LIN {X 0,Y 158.907,Z 446.881,A -85,B 0,C 180,E1 -23891.248,E2 -23891.248} C_VEL
LIN {X 0,Y 155.468,Z 440.852,A -85,B 0,C 180,E1 -23892.757,E2 -23892.757} C_VEL
LIN {X 0,Y 153.776,Z 436.815,A -85,B 0,C 180,E1 -23893.575,E2 -23893.575} C_VEL
LIN {X 0,Y 152.527,Z 433.767,A -85,B 0,C 180,E1 -23894.17,E2 -23894.17} C_VEL
LIN {X 0,Y 152.355,Z 432.875,A -85,B 0,C 180,E1 -23894.389,E2 -23894.389} C_VEL
LIN {X 0,Y 151.592,Z 429.44,A -85,B 0,C 180,E1 -23899.529,E2 -23899.529} C_VEL
LIN {X 0,Y 151.223,Z 427.382,A -85,B 0,C 180,E1 -23902.831,E2 -23902.831} C_VEL
LIN {X 0,Y 150.6,Z 423.714,A -85,B 0,C 180,E1 -23909.114,E2 -23909.114} C_VEL
LIN {X 0,Y 150.269,Z 421.77,A -85,B 0,C 180,E1 -23912.696,E2 -23912.696} C_VEL
LIN {X 0,Y 150.348,Z 421.758,A -85,B 0,C 180,E1 -23919.206,E2 -23919.206} C_VEL
LIN {X 0,Y 150.365,Z 421.755,A -85,B 0,C 180,E1 -23923.714,E2 -23923.714} C_VEL
LIN {X 0,Y 150.607,Z 421.725,A -85,B 0,C 180,E1 -23929.242,E2 -23929.242} C_VEL
LIN {X 0,Y 150.7,Z 421.71,A -85,B 0,C 180,E1 -23931.958,E2 -23931.958} C_VEL
LIN {X 0,Y 151.214,Z 421.648,A -85,B 0,C 180,E1 -23940,E2 -23940} C_VEL
LIN {X 0,Y 150.744,Z 421.707,A -85,B 0,C 180,E1 -23948.04,E2 -23948.04} C_VEL
LIN {X 0,Y 150.612,Z 421.713,A -85,B 0,C 180,E1 -23951.51,E2 -23951.51} C_VEL
LIN {X 0,Y 150.363,Z 421.751,A -85,B 0,C 180,E1 -23956.287,E2 -23956.287} C_VEL
LIN {X 0,Y 150.348,Z 421.749,A -85,B 0,C 180,E1 -23960.793,E2 -23960.793} C_VEL
LIN {X 0,Y 150.242,Z 421.769,A -85,B 0,C 180,E1 -23967.283,E2 -23967.283} C_VEL
LIN {X 0,Y 150.216,Z 421.758,A -85,B 0,C 180,E1 -23972.635,E2 -23972.635} C_VEL
LIN {X 0,Y 150.209,Z 421.774,A -85,B 0,C 180,E1 -23977.463,E2 -23977.463} C_VEL
LIN {X 0,Y 150.153,Z 421.767,A -85,B 0,C 180,E1 -23981.508,E2 -23981.508} C_VEL
LIN {X 0,Y 150.125,Z 421.785,A -85,B 0,C 180,E1 -23985.397,E2 -23985.397} C_VEL
LIN {X 0,Y 150.15,Z 421.764,A -85,B 0,C 180,E1 -23989.06,E2 -23989.06} C_VEL
LIN {X 0,Y 150.178,Z 421.737,A -85,B 0,C 180,E1 -23992.709,E2 -23992.709} C_VEL
LIN {X 0,Y 150.214,Z 421.775,A -85,B 0,C 180,E1 -23997.369,E2 -23997.369} C_VEL
LIN {X 0,Y 150.244,Z 421.752,A -85,B 0,C 180,E1 -24002.72,E2 -24002.72} C_VEL
LIN {X 0,Y 150.353,Z 421.757,A -85,B 0,C 180,E1 -24009.209,E2 -24009.209} C_VEL
LIN {X 0,Y 150.384,Z 421.737,A -85,B 0,C 180,E1 -24013.717,E2 -24013.717} C_VEL
LIN {X 0,Y 150.581,Z 421.722,A -85,B 0,C 180,E1 -24017.837,E2 -24017.837} C_VEL
LIN {X 0,Y 151.711,Z 424.669,A -85,B 0,C 180,E1 -24018.479,E2 -24018.479} C_VEL
LIN {X 0,Y 153.028,Z 426.654,A -85,B 0,C 180,E1 -24019.081,E2 -24019.081} C_VEL
LIN {X 0,Y 157.291,Z 435.385,A -85,B 0,C 180,E1 -24021.329,E2 -24021.329} C_VEL
LIN {X 0,Y 160.27,Z 442.518,A -85,B 0,C 180,E1 -24023.172,E2 -24023.172} C_VEL
LIN {X 0,Y 162.805,Z 453.417,A -85,B 0,C 180,E1 -24025.806,E2 -24025.806} C_VEL
LIN {X 0,Y 164.152,Z 461.495,A -85,B 0,C 180,E1 -24027.926,E2 -24027.926} C_VEL
LIN {X 0,Y 164.828,Z 468.949,A -85,B 0,C 180,E1 -24030.001,E2 -24030.001} C_VEL
LIN {X 0,Y 161.818,Z 479.094,A -85,B 0,C 180,E1 -24032.644,E2 -24032.644} C_VEL
LIN {X 0,Y 158.678,Z 488.449,A -85,B 0,C 180,E1 -24035.72,E2 -24035.72} C_VEL
LIN {X 0,Y 155.584,Z 497.087,A -85,B 0,C 180,E1 -24039.324,E2 -24039.324} C_VEL
LIN {X 0,Y 152.894,Z 504.421,A -85,B 0,C 180,E1 -24043.288,E2 -24043.288} C_VEL
LIN {X 0,Y 150.76,Z 510.595,A -85,B 0,C 180,E1 -24047.639,E2 -24047.639} C_VEL
LIN {X 0,Y 149.287,Z 515.38,A -85,B 0,C 180,E1 -24052.125,E2 -24052.125} C_VEL
LIN {X 0,Y 148.386,Z 518.306,A -85,B 0,C 180,E1 -24055.854,E2 -24055.854} C_VEL
LIN {X 0,Y 147.846,Z 521.083,A -85,B 0,C 180,E1 -24061.168,E2 -24061.168} C_VEL
LIN {X 0,Y 148.214,Z 522.273,A -85,B 0,C 180,E1 -24066.282,E2 -24066.282} C_VEL
LIN {X 0,Y 149.379,Z 522.141,A -85,B 0,C 180,E1 -24071.199,E2 -24071.199} C_VEL
LIN {X 0,Y 151.209,Z 520.831,A -85,B 0,C 180,E1 -24075.798,E2 -24075.798} C_VEL
LIN {X 0,Y 154.152,Z 517.931,A -85,B 0,C 180,E1 -24080.809,E2 -24080.809} C_VEL
LIN {X 0,Y 158.008,Z 513.502,A -85,B 0,C 180,E1 -24085.56,E2 -24085.56} C_VEL
LIN {X 0,Y 162.582,Z 507.7,A -85,B 0,C 180,E1 -24089.831,E2 -24089.831} C_VEL
LIN {X 0,Y 167.136,Z 501.227,A -85,B 0,C 180,E1 -24093.323,E2 -24093.323} C_VEL
LIN {X 0,Y 172.329,Z 492.969,A -85,B 0,C 180,E1 -24096.696,E2 -24096.696} C_VEL
LIN {X 0,Y 177.089,Z 484.362,A -85,B 0,C 180,E1 -24099.377,E2 -24099.377} C_VEL
LIN {X 0,Y 177.596,Z 476.445,A -85,B 0,C 180,E1 -24102.733,E2 -24102.733} C_VEL
LIN {X 0,Y 176.988,Z 469.941,A -85,B 0,C 180,E1 -24105.657,E2 -24105.657} C_VEL
LIN {X 0,Y 175.806,Z 464.39,A -85,B 0,C 180,E1 -24108.47,E2 -24108.47} C_VEL
LIN {X 0,Y 173.573,Z 458.192,A -85,B 0,C 180,E1 -24112.181,E2 -24112.181} C_VEL
LIN {X 0,Y 171.658,Z 453.679,A -85,B 0,C 180,E1 -24115.303,E2 -24115.303} C_VEL
LIN {X 0,Y 168.68,Z 447.648,A -85,B 0,C 180,E1 -24120.623,E2 -24120.623} C_VEL
LIN {X 0,Y 166.598,Z 444.818,A -85,B 0,C 180,E1 -24124.84,E2 -24124.84} C_VEL
LIN {X 0,Y 165.671,Z 443.784,A -85,B 0,C 180,E1 -24127.311,E2 -24127.311} C_VEL
LIN {X 0,Y 164.306,Z 443.346,A -85,B 0,C 180,E1 -24132.349,E2 -24132.349} C_VEL
LIN {X 0,Y 164.074,Z 444.083,A -85,B 0,C 180,E1 -24137.448,E2 -24137.448} C_VEL
LIN {X 0,Y 164.97,Z 446.098,A -85,B 0,C 180,E1 -24142.545,E2 -24142.545} C_VEL
LIN {X 0,Y 165.892,Z 447.367,A -85,B 0,C 180,E1 -24145.065,E2 -24145.065} C_VEL
LIN {X 0,Y 167.907,Z 452.872,A -85,B 0,C 180,E1 -24150.151,E2 -24150.151} C_VEL
LIN {X 0,Y 168.715,Z 453.994,A -85,B 0,C 180,E1 -24151.379,E2 -24151.379} C_VEL
LIN {X 0,Y 171.192,Z 460.649,A -85,B 0,C 180,E1 -24155.813,E2 -24155.813} C_VEL
LIN {X 0,Y 173.459,Z 467.717,A -85,B 0,C 180,E1 -24159.663,E2 -24159.663} C_VEL
LIN {X 0,Y 175.338,Z 474.627,A -85,B 0,C 180,E1 -24162.953,E2 -24162.953} C_VEL
LIN {X 0,Y 175.612,Z 476.996,A -85,B 0,C 180,E1 -24163.916,E2 -24163.916} C_VEL
LIN {X 0,Y 174.836,Z 486.166,A -85,B 0,C 180,E1 -24166.894,E2 -24166.894} C_VEL
LIN {X 0,Y 173.38,Z 494.259,A -85,B 0,C 180,E1 -24169.567,E2 -24169.567} C_VEL
LIN {X 0,Y 170.86,Z 503.046,A -85,B 0,C 180,E1 -24172.648,E2 -24172.648} C_VEL
LIN {X 0,Y 168.366,Z 509.152,A -85,B 0,C 180,E1 -24174.973,E2 -24174.973} C_VEL
LIN {X 0,Y 163.528,Z 517.051,A -85,B 0,C 180,E1 -24178.233,E2 -24178.233} C_VEL
LIN {X 0,Y 159.025,Z 523.782,A -85,B 0,C 180,E1 -24181.872,E2 -24181.872} C_VEL
LIN {X 0,Y 155.179,Z 529.387,A -85,B 0,C 180,E1 -24185.945,E2 -24185.945} C_VEL
LIN {X 0,Y 152.299,Z 533.334,A -85,B 0,C 180,E1 -24189.751,E2 -24189.751} C_VEL
LIN {X 0,Y 150.091,Z 536.305,A -85,B 0,C 180,E1 -24193.683,E2 -24193.683} C_VEL
LIN {X 0,Y 148.46,Z 538.834,A -85,B 0,C 180,E1 -24199.084,E2 -24199.084} C_VEL
LIN {X 0,Y 147.919,Z 539.85,A -85,B 0,C 180,E1 -24204.547,E2 -24204.547} C_VEL
LIN {X 0,Y 148.012,Z 539.745,A -85,B 0,C 180,E1 -24207.278,E2 -24207.278} C_VEL
LIN {X 0,Y 148.222,Z 539.247,A -85,B 0,C 180,E1 -24209.999,E2 -24209.999} C_VEL
LIN {X 0,Y 148.082,Z 537.369,A -85,B 0,C 180,E1 -24214.684,E2 -24214.684} C_VEL
LIN {X 0,Y 148.368,Z 534.065,A -85,B 0,C 180,E1 -24219.542,E2 -24219.542} C_VEL
LIN {X 0,Y 149.198,Z 530.096,A -85,B 0,C 180,E1 -24223.622,E2 -24223.622} C_VEL
LIN {X 0,Y 151.074,Z 523.962,A -85,B 0,C 180,E1 -24228.3,E2 -24228.3} C_VEL
LIN {X 0,Y 153.384,Z 517.248,A -85,B 0,C 180,E1 -24232.209,E2 -24232.209} C_VEL
LIN {X 0,Y 156.329,Z 508.999,A -85,B 0,C 180,E1 -24235.956,E2 -24235.956} C_VEL
LIN {X 0,Y 159.271,Z 500.325,A -85,B 0,C 180,E1 -24239.036,E2 -24239.036} C_VEL
LIN {X 0,Y 160.123,Z 493.994,A -85,B 0,C 180,E1 -24241.044,E2 -24241.044} C_VEL
LIN {X 0,Y 160.629,Z 484.356,A -85,B 0,C 180,E1 -24243.767,E2 -24243.767} C_VEL
LIN {X 0,Y 160.579,Z 473.096,A -85,B 0,C 180,E1 -24246.484,E2 -24246.484} C_VEL
LIN {X 0,Y 159.834,Z 461.563,A -85,B 0,C 180,E1 -24248.864,E2 -24248.864} C_VEL
LIN {X 0,Y 158.117,Z 448.898,A -85,B 0,C 180,E1 -24251.157,E2 -24251.157} C_VEL
LIN {X 0,Y 156.599,Z 443.784,A -85,B 0,C 180,E1 -24252.144,E2 -24252.144} C_VEL
LIN {X 0,Y 155.468,Z 440.852,A -85,B 0,C 180,E1 -24252.757,E2 -24252.757} C_VEL
LIN {X 0,Y 153.408,Z 437.999,A -85,B 0,C 180,E1 -24253.559,E2 -24253.559} C_VEL
LIN {X 0,Y 149.127,Z 434.501,A -85,B 0,C 180,E1 -24255.143,E2 -24255.143} C_VEL
LIN {X 0,Y 146.133,Z 432.507,A -85,B 0,C 180,E1 -24256.731,E2 -24256.731} C_VEL
LIN {X 0,Y 144.814,Z 431.33,A -85,B 0,C 180,E1 -24258.154,E2 -24258.154} C_VEL
LIN {X 0,Y 144.668,Z 430.996,A -85,B 0,C 180,E1 -24258.664,E2 -24258.664} C_VEL
LIN {X 0,Y 144.005,Z 427.728,A -85,B 0,C 180,E1 -24264.152,E2 -24264.152} C_VEL
LIN {X 0,Y 143.719,Z 425.864,A -85,B 0,C 180,E1 -24267.459,E2 -24267.459} C_VEL
LIN {X 0,Y 143.22,Z 422.805,A -85,B 0,C 180,E1 -24273.323,E2 -24273.323} C_VEL
LIN {X 0,Y 143.306,Z 422.634,A -85,B 0,C 180,E1 -24279.923,E2 -24279.923} C_VEL
LIN {X 0,Y 143.358,Z 422.627,A -85,B 0,C 180,E1 -24285.811,E2 -24285.811} C_VEL
LIN {X 0,Y 143.533,Z 422.606,A -85,B 0,C 180,E1 -24288.705,E2 -24288.705} C_VEL
LIN {X 0,Y 143.622,Z 422.592,A -85,B 0,C 180,E1 -24291.559,E2 -24291.559} C_VEL
LIN {X 0,Y 144.173,Z 422.525,A -85,B 0,C 180,E1 -24300,E2 -24300} C_VEL
LIN {X 0,Y 143.665,Z 422.59,A -85,B 0,C 180,E1 -24308.439,E2 -24308.439} C_VEL
LIN {X 0,Y 143.545,Z 422.591,A -85,B 0,C 180,E1 -24311.713,E2 -24311.713} C_VEL
LIN {X 0,Y 143.301,Z 422.634,A -85,B 0,C 180,E1 -24317.114,E2 -24317.114} C_VEL
LIN {X 0,Y 143.274,Z 422.627,A -85,B 0,C 180,E1 -24321.255,E2 -24321.255} C_VEL
LIN {X 0,Y 143.188,Z 422.649,A -85,B 0,C 180,E1 -24327.938,E2 -24327.938} C_VEL
LIN {X 0,Y 143.166,Z 422.638,A -85,B 0,C 180,E1 -24333.437,E2 -24333.437} C_VEL
LIN {X 0,Y 143.074,Z 422.654,A -85,B 0,C 180,E1 -24339.687,E2 -24339.687} C_VEL
LIN {X 0,Y 143.056,Z 422.662,A -85,B 0,C 180,E1 -24343.456,E2 -24343.456} C_VEL
LIN {X 0,Y 143.064,Z 422.659,A -85,B 0,C 180,E1 -24347.466,E2 -24347.466} C_VEL
LIN {X 0,Y 143.076,Z 422.621,A -85,B 0,C 180,E1 -24351.808,E2 -24351.808} C_VEL
LIN {X 0,Y 143.181,Z 422.651,A -85,B 0,C 180,E1 -24357.323,E2 -24357.323} C_VEL
LIN {X 0,Y 143.191,Z 422.636,A -85,B 0,C 180,E1 -24362.065,E2 -24362.065} C_VEL
LIN {X 0,Y 143.278,Z 422.638,A -85,B 0,C 180,E1 -24368.747,E2 -24368.747} C_VEL
LIN {X 0,Y 143.318,Z 422.614,A -85,B 0,C 180,E1 -24372.89,E2 -24372.89} C_VEL
LIN {X 0,Y 143.383,Z 422.626,A -85,B 0,C 180,E1 -24375.815,E2 -24375.815} C_VEL
LIN {X 0,Y 144.446,Z 425.514,A -85,B 0,C 180,E1 -24376.483,E2 -24376.483} C_VEL
LIN {X 0,Y 145.815,Z 427.401,A -85,B 0,C 180,E1 -24377.14,E2 -24377.14} C_VEL
LIN {X 0,Y 149.54,Z 434.414,A -85,B 0,C 180,E1 -24379.165,E2 -24379.165} C_VEL
LIN {X 0,Y 154.074,Z 444.914,A -85,B 0,C 180,E1 -24382.136,E2 -24382.136} C_VEL
LIN {X 0,Y 156.39,Z 455.339,A -85,B 0,C 180,E1 -24384.844,E2 -24384.844} C_VEL
LIN {X 0,Y 157.644,Z 462.899,A -85,B 0,C 180,E1 -24386.976,E2 -24386.976} C_VEL
LIN {X 0,Y 158.234,Z 469.919,A -85,B 0,C 180,E1 -24389.046,E2 -24389.046} C_VEL
LIN {X 0,Y 155.349,Z 479.333,A -85,B 0,C 180,E1 -24391.597,E2 -24391.597} C_VEL
LIN {X 0,Y 152.223,Z 488.325,A -85,B 0,C 180,E1 -24394.635,E2 -24394.635} C_VEL
LIN {X 0,Y 149.1,Z 496.612,A -85,B 0,C 180,E1 -24398.163,E2 -24398.163} C_VEL
LIN {X 0,Y 146.581,Z 503.279,A -85,B 0,C 180,E1 -24401.758,E2 -24401.758} C_VEL
LIN {X 0,Y 144.498,Z 508.9,A -85,B 0,C 180,E1 -24405.574,E2 -24405.574} C_VEL
LIN {X 0,Y 142.586,Z 514.475,A -85,B 0,C 180,E1 -24410.527,E2 -24410.527} C_VEL
LIN {X 0,Y 141.481,Z 518.034,A -85,B 0,C 180,E1 -24414.846,E2 -24414.846} C_VEL
LIN {X 0,Y 140.778,Z 520.893,A -85,B 0,C 180,E1 -24419.949,E2 -24419.949} C_VEL
LIN {X 0,Y 140.786,Z 522.087,A -85,B 0,C 180,E1 -24423.307,E2 -24423.307} C_VEL
LIN {X 0,Y 141.28,Z 522.757,A -85,B 0,C 180,E1 -24427.257,E2 -24427.257} C_VEL
LIN {X 0,Y 142.618,Z 522.557,A -85,B 0,C 180,E1 -24432.338,E2 -24432.338} C_VEL
LIN {X 0,Y 144.701,Z 521.173,A -85,B 0,C 180,E1 -24437.158,E2 -24437.158} C_VEL
LIN {X 0,Y 147.499,Z 518.658,A -85,B 0,C 180,E1 -24441.726,E2 -24441.726} C_VEL
LIN {X 0,Y 151.551,Z 514.407,A -85,B 0,C 180,E1 -24446.587,E2 -24446.587} C_VEL
LIN {X 0,Y 155.308,Z 510.019,A -85,B 0,C 180,E1 -24450.147,E2 -24450.147} C_VEL
LIN {X 0,Y 160.333,Z 503.604,A -85,B 0,C 180,E1 -24454.002,E2 -24454.002} C_VEL
LIN {X 0,Y 165.827,Z 495.604,A -85,B 0,C 180,E1 -24457.577,E2 -24457.577} C_VEL
LIN {X 0,Y 171.331,Z 486.46,A -85,B 0,C 180,E1 -24460.64,E2 -24460.64} C_VEL
LIN {X 0,Y 172.029,Z 480.432,A -85,B 0,C 180,E1 -24463.383,E2 -24463.383} C_VEL
LIN {X 0,Y 171.831,Z 474.271,A -85,B 0,C 180,E1 -24466.398,E2 -24466.398} C_VEL
LIN {X 0,Y 170.941,Z 468.915,A -85,B 0,C 180,E1 -24469.338,E2 -24469.338} C_VEL
LIN {X 0,Y 169.311,Z 463.496,A -85,B 0,C 180,E1 -24472.846,E2 -24472.846} C_VEL
LIN {X 0,Y 167.569,Z 458.742,A -85,B 0,C 180,E1 -24476.438,E2 -24476.438} C_VEL
LIN {X 0,Y 165.884,Z 454.97,A -85,B 0,C 180,E1 -24480,E2 -24480} C_VEL
LIN {X 0,Y 163.881,Z 451.424,A -85,B 0,C 180,E1 -24484.92,E2 -24484.92} C_VEL
LIN {X 0,Y 163.035,Z 450.369,A -85,B 0,C 180,E1 -24487.493,E2 -24487.493} C_VEL
LIN {X 0,Y 161.793,Z 450.007,A -85,B 0,C 180,E1 -24492.544,E2 -24492.544} C_VEL
LIN {X 0,Y 161.615,Z 450.834,A -85,B 0,C 180,E1 -24497.722,E2 -24497.722} C_VEL
LIN {X 0,Y 162.51,Z 452.951,A -85,B 0,C 180,E1 -24502.906,E2 -24502.906} C_VEL
LIN {X 0,Y 163.318,Z 454.588,A -85,B 0,C 180,E1 -24505.488,E2 -24505.488} C_VEL
LIN {X 0,Y 164.54,Z 458.78,A -85,B 0,C 180,E1 -24509.419,E2 -24509.419} C_VEL
LIN {X 0,Y 165.247,Z 459.919,A -85,B 0,C 180,E1 -24510.688,E2 -24510.688} C_VEL
LIN {X 0,Y 167.199,Z 466.143,A -85,B 0,C 180,E1 -24515.102,E2 -24515.102} C_VEL
LIN {X 0,Y 169.094,Z 473.233,A -85,B 0,C 180,E1 -24519.206,E2 -24519.206} C_VEL
LIN {X 0,Y 170.287,Z 478.763,A -85,B 0,C 180,E1 -24522.022,E2 -24522.022} C_VEL
LIN {X 0,Y 170.335,Z 481.66,A -85,B 0,C 180,E1 -24523.213,E2 -24523.213} C_VEL
LIN {X 0,Y 168.973,Z 490.428,A -85,B 0,C 180,E1 -24526.28,E2 -24526.28} C_VEL
LIN {X 0,Y 166.815,Z 498.905,A -85,B 0,C 180,E1 -24529.319,E2 -24529.319} C_VEL
LIN {X 0,Y 163.92,Z 506.738,A -85,B 0,C 180,E1 -24532.341,E2 -24532.341} C_VEL
LIN {X 0,Y 160.952,Z 512.325,A -85,B 0,C 180,E1 -24534.65,E2 -24534.65} C_VEL
LIN {X 0,Y 155.946,Z 519.549,A -85,B 0,C 180,E1 -24538.026,E2 -24538.026} C_VEL
LIN {X 0,Y 151.107,Z 526.257,A -85,B 0,C 180,E1 -24542.283,E2 -24542.283} C_VEL
LIN {X 0,Y 147.579,Z 530.777,A -85,B 0,C 180,E1 -24546.122,E2 -24546.122} C_VEL
LIN {X 0,Y 144.764,Z 534.281,A -85,B 0,C 180,E1 -24550.133,E2 -24550.133} C_VEL
LIN {X 0,Y 142.195,Z 537.473,A -85,B 0,C 180,E1 -24555.692,E2 -24555.692} C_VEL
LIN {X 0,Y 141.002,Z 539.157,A -85,B 0,C 180,E1 -24561.4,E2 -24561.4} C_VEL
LIN {X 0,Y 140.869,Z 539.355,A -85,B 0,C 180,E1 -24566.205,E2 -24566.205} C_VEL
LIN {X 0,Y 141.159,Z 538.704,A -85,B 0,C 180,E1 -24569.999,E2 -24569.999} C_VEL
LIN {X 0,Y 141.016,Z 536.892,A -85,B 0,C 180,E1 -24574.609,E2 -24574.609} C_VEL
LIN {X 0,Y 141.343,Z 533.316,A -85,B 0,C 180,E1 -24580.021,E2 -24580.021} C_VEL
LIN {X 0,Y 142.258,Z 529.247,A -85,B 0,C 180,E1 -24584.3,E2 -24584.3} C_VEL
LIN {X 0,Y 144.33,Z 522.995,A -85,B 0,C 180,E1 -24589.188,E2 -24589.188} C_VEL
LIN {X 0,Y 146.814,Z 516.166,A -85,B 0,C 180,E1 -24593.26,E2 -24593.26} C_VEL
LIN {X 0,Y 149.593,Z 508.618,A -85,B 0,C 180,E1 -24596.794,E2 -24596.794} C_VEL
LIN {X 0,Y 152.398,Z 500.792,A -85,B 0,C 180,E1 -24599.718,E2 -24599.718} C_VEL
LIN {X 0,Y 153.24,Z 495.687,A -85,B 0,C 180,E1 -24601.444,E2 -24601.444} C_VEL
LIN {X 0,Y 153.947,Z 485.519,A -85,B 0,C 180,E1 -24604.519,E2 -24604.519} C_VEL
LIN {X 0,Y 154.056,Z 473.769,A -85,B 0,C 180,E1 -24607.545,E2 -24607.545} C_VEL
LIN {X 0,Y 153.472,Z 462.291,A -85,B 0,C 180,E1 -24610.086,E2 -24610.086} C_VEL
LIN {X 0,Y 151.971,Z 450.6,A -85,B 0,C 180,E1 -24612.384,E2 -24612.384} C_VEL
LIN {X 0,Y 149.75,Z 444.072,A -85,B 0,C 180,E1 -24613.816,E2 -24613.816} C_VEL
LIN {X 0,Y 146.543,Z 436.41,A -85,B 0,C 180,E1 -24615.552,E2 -24615.552} C_VEL
LIN {X 0,Y 145.151,Z 433.181,A -85,B 0,C 180,E1 -24616.27,E2 -24616.27} C_VEL
LIN {X 0,Y 144.998,Z 432.363,A -85,B 0,C 180,E1 -24616.452,E2 -24616.452} C_VEL
LIN {X 0,Y 144.668,Z 430.996,A -85,B 0,C 180,E1 -24618.664,E2 -24618.664} C_VEL
LIN {X 0,Y 143.741,Z 429.741,A -85,B 0,C 180,E1 -24620.919,E2 -24620.919} C_VEL
LIN {X 0,Y 141.888,Z 428.673,A -85,B 0,C 180,E1 -24623.144,E2 -24623.144} C_VEL
LIN {X 0,Y 137.702,Z 426.762,A -85,B 0,C 180,E1 -24627.709,E2 -24627.709} C_VEL
LIN {X 0,Y 136.531,Z 425.689,A -85,B 0,C 180,E1 -24630.132,E2 -24630.132} C_VEL
LIN {X 0,Y 136.43,Z 425.287,A -85,B 0,C 180,E1 -24630.954,E2 -24630.954} C_VEL
LIN {X 0,Y 136.107,Z 423.532,A -85,B 0,C 180,E1 -24634.786,E2 -24634.786} C_VEL
LIN {X 0,Y 136.241,Z 423.515,A -85,B 0,C 180,E1 -24638.833,E2 -24638.833} C_VEL
LIN {X 0,Y 136.268,Z 423.511,A -85,B 0,C 180,E1 -24645.056,E2 -24645.056} C_VEL
LIN {X 0,Y 136.441,Z 423.489,A -85,B 0,C 180,E1 -24648.138,E2 -24648.138} C_VEL
LIN {X 0,Y 136.547,Z 423.474,A -85,B 0,C 180,E1 -24651.118,E2 -24651.118} C_VEL
LIN {X 0,Y 137.13,Z 423.402,A -85,B 0,C 180,E1 -24660,E2 -24660} C_VEL
LIN {X 0,Y 136.591,Z 423.469,A -85,B 0,C 180,E1 -24668.88,E2 -24668.88} C_VEL
LIN {X 0,Y 136.488,Z 423.467,A -85,B 0,C 180,E1 -24671.955,E2 -24671.955} C_VEL
LIN {X 0,Y 136.241,Z 423.514,A -85,B 0,C 180,E1 -24678.03,E2 -24678.03} C_VEL
LIN {X 0,Y 136.195,Z 423.505,A -85,B 0,C 180,E1 -24681.749,E2 -24681.749} C_VEL
LIN {X 0,Y 136.098,Z 423.531,A -85,B 0,C 180,E1 -24688.618,E2 -24688.618} C_VEL
LIN {X 0,Y 136.077,Z 423.527,A -85,B 0,C 180,E1 -24694.62,E2 -24694.62} C_VEL
LIN {X 0,Y 136.049,Z 423.532,A -85,B 0,C 180,E1 -24699.21,E2 -24699.21} C_VEL
LIN {X 0,Y 135.997,Z 423.542,A -85,B 0,C 180,E1 -24703.659,E2 -24703.659} C_VEL
LIN {X 0,Y 136.004,Z 423.535,A -85,B 0,C 180,E1 -24707.798,E2 -24707.798} C_VEL
LIN {X 0,Y 136.025,Z 423.498,A -85,B 0,C 180,E1 -24711.685,E2 -24711.685} C_VEL
LIN {X 0,Y 136.054,Z 423.521,A -85,B 0,C 180,E1 -24715.741,E2 -24715.741} C_VEL
LIN {X 0,Y 136.147,Z 423.509,A -85,B 0,C 180,E1 -24722.318,E2 -24722.318} C_VEL
LIN {X 0,Y 136.245,Z 423.515,A -85,B 0,C 180,E1 -24728.834,E2 -24728.834} C_VEL
LIN {X 0,Y 136.287,Z 423.578,A -85,B 0,C 180,E1 -24733.573,E2 -24733.573} C_VEL
LIN {X 0,Y 137.182,Z 426.211,A -85,B 0,C 180,E1 -24734.2,E2 -24734.2} C_VEL
LIN {X 0,Y 138.71,Z 428.353,A -85,B 0,C 180,E1 -24735.024,E2 -24735.024} C_VEL
LIN {X 0,Y 143.7,Z 437.421,A -85,B 0,C 180,E1 -24738.002,E2 -24738.002} C_VEL
LIN {X 0,Y 147.807,Z 447.336,A -85,B 0,C 180,E1 -24741.013,E2 -24741.013} C_VEL
LIN {X 0,Y 149.107,Z 452.521,A -85,B 0,C 180,E1 -24742.487,E2 -24742.487} C_VEL
LIN {X 0,Y 151.025,Z 463.223,A -85,B 0,C 180,E1 -24745.648,E2 -24745.648} C_VEL
LIN {X 0,Y 151.645,Z 470.789,A -85,B 0,C 180,E1 -24748.009,E2 -24748.009} C_VEL
LIN {X 0,Y 148.894,Z 479.611,A -85,B 0,C 180,E1 -24750.502,E2 -24750.502} C_VEL
LIN {X 0,Y 145.113,Z 489.92,A -85,B 0,C 180,E1 -24754.167,E2 -24754.167} C_VEL
LIN {X 0,Y 141.904,Z 498.066,A -85,B 0,C 180,E1 -24757.889,E2 -24757.889} C_VEL
LIN {X 0,Y 139.338,Z 504.522,A -85,B 0,C 180,E1 -24761.64,E2 -24761.64} C_VEL
LIN {X 0,Y 136.918,Z 510.849,A -85,B 0,C 180,E1 -24766.399,E2 -24766.399} C_VEL
LIN {X 0,Y 135.231,Z 515.774,A -85,B 0,C 180,E1 -24771.334,E2 -24771.334} C_VEL
LIN {X 0,Y 133.997,Z 519.738,A -85,B 0,C 180,E1 -24776.919,E2 -24776.919} C_VEL
LIN {X 0,Y 133.669,Z 522.218,A -85,B 0,C 180,E1 -24782.727,E2 -24782.727} C_VEL
LIN {X 0,Y 134.481,Z 523.284,A -85,B 0,C 180,E1 -24788.838,E2 -24788.838} C_VEL
LIN {X 0,Y 135.927,Z 522.972,A -85,B 0,C 180,E1 -24793.625,E2 -24793.625} C_VEL
LIN {X 0,Y 138.277,Z 521.515,A -85,B 0,C 180,E1 -24798.644,E2 -24798.644} C_VEL
LIN {X 0,Y 141.378,Z 518.931,A -85,B 0,C 180,E1 -24803.378,E2 -24803.378} C_VEL
LIN {X 0,Y 145.274,Z 515.17,A -85,B 0,C 180,E1 -24807.848,E2 -24807.848} C_VEL
LIN {X 0,Y 149.986,Z 510.114,A -85,B 0,C 180,E1 -24812.058,E2 -24812.058} C_VEL
LIN {X 0,Y 155.315,Z 503.681,A -85,B 0,C 180,E1 -24815.967,E2 -24815.967} C_VEL
LIN {X 0,Y 160.046,Z 497.245,A -85,B 0,C 180,E1 -24818.92,E2 -24818.92} C_VEL
LIN {X 0,Y 165.581,Z 488.714,A -85,B 0,C 180,E1 -24821.928,E2 -24821.928} C_VEL
LIN {X 0,Y 166.501,Z 483.071,A -85,B 0,C 180,E1 -24824.703,E2 -24824.703} C_VEL
LIN {X 0,Y 166.558,Z 477.261,A -85,B 0,C 180,E1 -24827.82,E2 -24827.82} C_VEL
LIN {X 0,Y 165.587,Z 471.537,A -85,B 0,C 180,E1 -24831.457,E2 -24831.457} C_VEL
LIN {X 0,Y 164.302,Z 466.621,A -85,B 0,C 180,E1 -24835.092,E2 -24835.092} C_VEL
LIN {X 0,Y 162.862,Z 462.655,A -85,B 0,C 180,E1 -24838.763,E2 -24838.763} C_VEL
LIN {X 0,Y 161.74,Z 459.839,A -85,B 0,C 180,E1 -24841.987,E2 -24841.987} C_VEL
LIN {X 0,Y 160.804,Z 457.866,A -85,B 0,C 180,E1 -24845.014,E2 -24845.014} C_VEL
LIN {X 0,Y 160.098,Z 456.836,A -85,B 0,C 180,E1 -24847.567,E2 -24847.567} C_VEL
LIN {X 0,Y 158.86,Z 456.595,A -85,B 0,C 180,E1 -24853.276,E2 -24853.276} C_VEL
LIN {X 0,Y 158.787,Z 457.498,A -85,B 0,C 180,E1 -24858.048,E2 -24858.048} C_VEL
LIN {X 0,Y 159.676,Z 459.755,A -85,B 0,C 180,E1 -24863.336,E2 -24863.336} C_VEL
LIN {X 0,Y 160.121,Z 460.829,A -85,B 0,C 180,E1 -24865.019,E2 -24865.019} C_VEL
LIN {X 0,Y 161.198,Z 465.113,A -85,B 0,C 180,E1 -24869.313,E2 -24869.313} C_VEL
LIN {X 0,Y 161.537,Z 465.697,A -85,B 0,C 180,E1 -24870.02,E2 -24870.02} C_VEL
LIN {X 0,Y 162.927,Z 471.062,A -85,B 0,C 180,E1 -24874.109,E2 -24874.109} C_VEL
LIN {X 0,Y 164.422,Z 478.274,A -85,B 0,C 180,E1 -24878.57,E2 -24878.57} C_VEL
LIN {X 0,Y 165.158,Z 483.197,A -85,B 0,C 180,E1 -24881.266,E2 -24881.266} C_VEL
LIN {X 0,Y 164.917,Z 485.89,A -85,B 0,C 180,E1 -24882.388,E2 -24882.388} C_VEL
LIN {X 0,Y 162.968,Z 494.608,A -85,B 0,C 180,E1 -24885.681,E2 -24885.681} C_VEL
LIN {X 0,Y 160.25,Z 502.748,A -85,B 0,C 180,E1 -24888.864,E2 -24888.864} C_VEL
LIN {X 0,Y 156.871,Z 510.117,A -85,B 0,C 180,E1 -24891.974,E2 -24891.974} C_VEL
LIN {X 0,Y 152.537,Z 516.472,A -85,B 0,C 180,E1 -24894.836,E2 -24894.836} C_VEL
LIN {X 0,Y 147.607,Z 522.795,A -85,B 0,C 180,E1 -24898.416,E2 -24898.416} C_VEL
LIN {X 0,Y 143.569,Z 527.914,A -85,B 0,C 180,E1 -24902.287,E2 -24902.287} C_VEL
LIN {X 0,Y 139.995,Z 531.976,A -85,B 0,C 180,E1 -24906.321,E2 -24906.321} C_VEL
LIN {X 0,Y 136.445,Z 535.845,A -85,B 0,C 180,E1 -24911.998,E2 -24911.998} C_VEL
LIN {X 0,Y 134.474,Z 538.18,A -85,B 0,C 180,E1 -24917.933,E2 -24917.933} C_VEL
LIN {X 0,Y 133.756,Z 538.932,A -85,B 0,C 180,E1 -24923.967,E2 -24923.967} C_VEL
LIN {X 0,Y 133.845,Z 538.74,A -85,B 0,C 180,E1 -24926.989,E2 -24926.989} C_VEL
LIN {X 0,Y 134.095,Z 538.16,A -85,B 0,C 180,E1 -24929.999,E2 -24929.999} C_VEL
LIN {X 0,Y 133.947,Z 536.418,A -85,B 0,C 180,E1 -24934.512,E2 -24934.512} C_VEL
LIN {X 0,Y 134.345,Z 532.536,A -85,B 0,C 180,E1 -24940.549,E2 -24940.549} C_VEL
LIN {X 0,Y 135.354,Z 528.363,A -85,B 0,C 180,E1 -24945.046,E2 -24945.046} C_VEL
LIN {X 0,Y 137.625,Z 522.003,A -85,B 0,C 180,E1 -24950.162,E2 -24950.162} C_VEL
LIN {X 0,Y 140.294,Z 515.04,A -85,B 0,C 180,E1 -24954.41,E2 -24954.41} C_VEL
LIN {X 0,Y 142.971,Z 508.048,A -85,B 0,C 180,E1 -24957.771,E2 -24957.771} C_VEL
LIN {X 0,Y 146.091,Z 499.265,A -85,B 0,C 180,E1 -24961.14,E2 -24961.14} C_VEL
LIN {X 0,Y 147.008,Z 490.435,A -85,B 0,C 180,E1 -24964.174,E2 -24964.174} C_VEL
LIN {X 0,Y 147.501,Z 480.44,A -85,B 0,C 180,E1 -24967.126,E2 -24967.126} C_VEL
LIN {X 0,Y 147.451,Z 469.381,A -85,B 0,C 180,E1 -24969.935,E2 -24969.935} C_VEL
LIN {X 0,Y 146.523,Z 456.779,A -85,B 0,C 180,E1 -24972.723,E2 -24972.723} C_VEL
LIN {X 0,Y 145.79,Z 452.173,A -85,B 0,C 180,E1 -24973.689,E2 -24973.689} C_VEL
LIN {X 0,Y 142.392,Z 443.039,A -85,B 0,C 180,E1 -24975.982,E2 -24975.982} C_VEL
LIN {X 0,Y 139.406,Z 436.276,A -85,B 0,C 180,E1 -24977.724,E2 -24977.724} C_VEL
LIN {X 0,Y 137.939,Z 433.247,A -85,B 0,C 180,E1 -24978.521,E2 -24978.521} C_VEL
LIN {X 0,Y 137.655,Z 431.918,A -85,B 0,C 180,E1 -24978.798,E2 -24978.798} C_VEL
LIN {X 0,Y 136.861,Z 428.038,A -85,B 0,C 180,E1 -24985.607,E2 -24985.607} C_VEL
LIN {X 0,Y 136.43,Z 425.287,A -85,B 0,C 180,E1 -24990.954,E2 -24990.954} C_VEL
LIN {X 0,Y 135.724,Z 424.399,A -85,B 0,C 180,E1 -24993.379,E2 -24993.379} C_VEL
LIN {X 0,Y 134.116,Z 424.051,A -85,B 0,C 180,E1 -24995.798,E2 -24995.798} C_VEL
LIN {X 0,Y 129.524,Z 424.355,A -85,B 0,C 180,E1 -25002.517,E2 -25002.517} C_VEL
LIN {X 0,Y 129.192,Z 424.392,A -85,B 0,C 180,E1 -25004.298,E2 -25004.298} C_VEL
LIN {X 0,Y 129.363,Z 424.371,A -85,B 0,C 180,E1 -25007.922,E2 -25007.922} C_VEL
LIN {X 0,Y 129.473,Z 424.358,A -85,B 0,C 180,E1 -25010.628,E2 -25010.628} C_VEL
LIN {X 0,Y 130.085,Z 424.279,A -85,B 0,C 180,E1 -25020,E2 -25020} C_VEL
LIN {X 0,Y 129.516,Z 424.35,A -85,B 0,C 180,E1 -25029.369,E2 -25029.369} C_VEL
LIN {X 0,Y 129.39,Z 424.348,A -85,B 0,C 180,E1 -25032.549,E2 -25032.549} C_VEL
LIN {X 0,Y 129.151,Z 424.396,A -85,B 0,C 180,E1 -25039.057,E2 -25039.057} C_VEL
LIN {X 0,Y 129.106,Z 424.384,A -85,B 0,C 180,E1 -25042.399,E2 -25042.399} C_VEL
LIN {X 0,Y 129.033,Z 424.409,A -85,B 0,C 180,E1 -25049.374,E2 -25049.374} C_VEL
LIN {X 0,Y 128.991,Z 424.414,A -85,B 0,C 180,E1 -25055.191,E2 -25055.191} C_VEL
LIN {X 0,Y 128.949,Z 424.407,A -85,B 0,C 180,E1 -25060.846,E2 -25060.846} C_VEL
LIN {X 0,Y 128.92,Z 424.427,A -85,B 0,C 180,E1 -25065.129,E2 -25065.129} C_VEL
LIN {X 0,Y 128.941,Z 424.394,A -85,B 0,C 180,E1 -25069.737,E2 -25069.737} C_VEL
LIN {X 0,Y 128.957,Z 424.391,A -85,B 0,C 180,E1 -25074.834,E2 -25074.834} C_VEL
LIN {X 0,Y 129.034,Z 424.411,A -85,B 0,C 180,E1 -25080.648,E2 -25080.648} C_VEL
LIN {X 0,Y 129.109,Z 424.397,A -85,B 0,C 180,E1 -25087.603,E2 -25087.603} C_VEL
LIN {X 0,Y 129.201,Z 424.566,A -85,B 0,C 180,E1 -25091.051,E2 -25091.051} C_VEL
LIN {X 0,Y 130.134,Z 427.106,A -85,B 0,C 180,E1 -25091.768,E2 -25091.768} C_VEL
LIN {X 0,Y 131.635,Z 429.221,A -85,B 0,C 180,E1 -25092.663,E2 -25092.663} C_VEL
LIN {X 0,Y 133.466,Z 432.413,A -85,B 0,C 180,E1 -25093.828,E2 -25093.828} C_VEL
LIN {X 0,Y 137.938,Z 440.686,A -85,B 0,C 180,E1 -25096.824,E2 -25096.824} C_VEL
LIN {X 0,Y 141.529,Z 449.562,A -85,B 0,C 180,E1 -25099.796,E2 -25099.796} C_VEL
LIN {X 0,Y 142.723,Z 453.61,A -85,B 0,C 180,E1 -25101.084,E2 -25101.084} C_VEL
LIN {X 0,Y 144.553,Z 464.254,A -85,B 0,C 180,E1 -25104.421,E2 -25104.421} C_VEL
LIN {X 0,Y 144.982,Z 472.721,A -85,B 0,C 180,E1 -25107.222,E2 -25107.222} C_VEL
LIN {X 0,Y 141.148,Z 483.524,A -85,B 0,C 180,E1 -25110.528,E2 -25110.528} C_VEL
LIN {X 0,Y 137.317,Z 493.156,A -85,B 0,C 180,E1 -25114.404,E2 -25114.404} C_VEL
LIN {X 0,Y 134.297,Z 500.513,A -85,B 0,C 180,E1 -25118.204,E2 -25118.204} C_VEL
LIN {X 0,Y 131.666,Z 506.825,A -85,B 0,C 180,E1 -25122.329,E2 -25122.329} C_VEL
LIN {X 0,Y 129.275,Z 512.811,A -85,B 0,C 180,E1 -25127.398,E2 -25127.398} C_VEL
LIN {X 0,Y 127.742,Z 517.35,A -85,B 0,C 180,E1 -25132.652,E2 -25132.652} C_VEL
LIN {X 0,Y 126.794,Z 520.388,A -85,B 0,C 180,E1 -25137.518,E2 -25137.518} C_VEL
LIN {X 0,Y 126.622,Z 522.796,A -85,B 0,C 180,E1 -25143.714,E2 -25143.714} C_VEL
LIN {X 0,Y 127.508,Z 523.723,A -85,B 0,C 180,E1 -25149.496,E2 -25149.496} C_VEL
LIN {X 0,Y 129.334,Z 523.37,A -85,B 0,C 180,E1 -25155.055,E2 -25155.055} C_VEL
LIN {X 0,Y 131.985,Z 521.838,A -85,B 0,C 180,E1 -25160.283,E2 -25160.283} C_VEL
LIN {X 0,Y 135.919,Z 518.773,A -85,B 0,C 180,E1 -25165.824,E2 -25165.824} C_VEL
LIN {X 0,Y 141.009,Z 514.148,A -85,B 0,C 180,E1 -25171.011,E2 -25171.011} C_VEL
LIN {X 0,Y 146.712,Z 508.147,A -85,B 0,C 180,E1 -25175.527,E2 -25175.527} C_VEL
LIN {X 0,Y 152.267,Z 501.505,A -85,B 0,C 180,E1 -25179.171,E2 -25179.171} C_VEL
LIN {X 0,Y 158.601,Z 492.902,A -85,B 0,C 180,E1 -25182.652,E2 -25182.652} C_VEL
LIN {X 0,Y 160.063,Z 490.687,A -85,B 0,C 180,E1 -25183.418,E2 -25183.418} C_VEL
LIN {X 0,Y 161.063,Z 485.535,A -85,B 0,C 180,E1 -25186.203,E2 -25186.203} C_VEL
LIN {X 0,Y 161.29,Z 481.294,A -85,B 0,C 180,E1 -25188.692,E2 -25188.692} C_VEL
LIN {X 0,Y 160.674,Z 475.932,A -85,B 0,C 180,E1 -25192.459,E2 -25192.459} C_VEL
LIN {X 0,Y 159.759,Z 471.352,A -85,B 0,C 180,E1 -25196.216,E2 -25196.216} C_VEL
LIN {X 0,Y 158.678,Z 467.647,A -85,B 0,C 180,E1 -25200,E2 -25200} C_VEL
LIN {X 0,Y 157.998,Z 465.68,A -85,B 0,C 180,E1 -25202.549,E2 -25202.549} C_VEL
LIN {X 0,Y 157.37,Z 464.105,A -85,B 0,C 180,E1 -25205.124,E2 -25205.124} C_VEL
LIN {X 0,Y 156.804,Z 463.107,A -85,B 0,C 180,E1 -25207.727,E2 -25207.727} C_VEL
LIN {X 0,Y 155.737,Z 462.912,A -85,B 0,C 180,E1 -25213.04,E2 -25213.04} C_VEL
LIN {X 0,Y 155.621,Z 464.039,A -85,B 0,C 180,E1 -25218.491,E2 -25218.491} C_VEL
LIN {X 0,Y 155.945,Z 465.031,A -85,B 0,C 180,E1 -25221.133,E2 -25221.133} C_VEL
LIN {X 0,Y 156.465,Z 466.437,A -85,B 0,C 180,E1 -25223.844,E2 -25223.844} C_VEL
LIN {X 0,Y 157.598,Z 471.377,A -85,B 0,C 180,E1 -25229.376,E2 -25229.376} C_VEL
LIN {X 0,Y 158.754,Z 477.709,A -85,B 0,C 180,E1 -25234.362,E2 -25234.362} C_VEL
LIN {X 0,Y 159.77,Z 484.933,A -85,B 0,C 180,E1 -25239.059,E2 -25239.059} C_VEL
LIN {X 0,Y 159.869,Z 487.905,A -85,B 0,C 180,E1 -25240.688,E2 -25240.688} C_VEL
LIN {X 0,Y 157.752,Z 495.71,A -85,B 0,C 180,E1 -25243.85,E2 -25243.85} C_VEL
LIN {X 0,Y 154.857,Z 503.463,A -85,B 0,C 180,E1 -25247.097,E2 -25247.097} C_VEL
LIN {X 0,Y 151.278,Z 510.579,A -85,B 0,C 180,E1 -25250.298,E2 -25250.298} C_VEL
LIN {X 0,Y 147.721,Z 515.633,A -85,B 0,C 180,E1 -25252.656,E2 -25252.656} C_VEL
LIN {X 0,Y 143.259,Z 521.037,A -85,B 0,C 180,E1 -25255.656,E2 -25255.656} C_VEL
LIN {X 0,Y 138.614,Z 526.402,A -85,B 0,C 180,E1 -25259.534,E2 -25259.534} C_VEL
LIN {X 0,Y 134.686,Z 530.668,A -85,B 0,C 180,E1 -25263.67,E2 -25263.67} C_VEL
LIN {X 0,Y 131.443,Z 533.945,A -85,B 0,C 180,E1 -25268.02,E2 -25268.02} C_VEL
LIN {X 0,Y 128.416,Z 536.932,A -85,B 0,C 180,E1 -25274.118,E2 -25274.118} C_VEL
LIN {X 0,Y 126.927,Z 538.332,A -85,B 0,C 180,E1 -25280.438,E2 -25280.438} C_VEL
LIN {X 0,Y 126.768,Z 538.232,A -85,B 0,C 180,E1 -25286.821,E2 -25286.821} C_VEL
LIN {X 0,Y 127.032,Z 537.605,A -85,B 0,C 180,E1 -25289.999,E2 -25289.999} C_VEL
LIN {X 0,Y 126.879,Z 535.935,A -85,B 0,C 180,E1 -25294.405,E2 -25294.405} C_VEL
LIN {X 0,Y 127.346,Z 531.749,A -85,B 0,C 180,E1 -25301.136,E2 -25301.136} C_VEL
LIN {X 0,Y 128.481,Z 527.473,A -85,B 0,C 180,E1 -25305.872,E2 -25305.872} C_VEL
LIN {X 0,Y 130.945,Z 521.001,A -85,B 0,C 180,E1 -25311.239,E2 -25311.239} C_VEL
LIN {X 0,Y 133.826,Z 513.859,A -85,B 0,C 180,E1 -25315.673,E2 -25315.673} C_VEL
LIN {X 0,Y 136.809,Z 506.434,A -85,B 0,C 180,E1 -25319.289,E2 -25319.289} C_VEL
LIN {X 0,Y 139.304,Z 499.691,A -85,B 0,C 180,E1 -25321.986,E2 -25321.986} C_VEL
LIN {X 0,Y 140.347,Z 490.993,A -85,B 0,C 180,E1 -25325.159,E2 -25325.159} C_VEL
LIN {X 0,Y 140.958,Z 481.674,A -85,B 0,C 180,E1 -25328.094,E2 -25328.094} C_VEL
LIN {X 0,Y 141.092,Z 471.289,A -85,B 0,C 180,E1 -25330.936,E2 -25330.936} C_VEL
LIN {X 0,Y 140.569,Z 460.518,A -85,B 0,C 180,E1 -25333.537,E2 -25333.537} C_VEL
LIN {X 0,Y 140.041,Z 455.743,A -85,B 0,C 180,E1 -25334.633,E2 -25334.633} C_VEL
LIN {X 0,Y 136.371,Z 444.967,A -85,B 0,C 180,E1 -25337.562,E2 -25337.562} C_VEL
LIN {X 0,Y 132.736,Z 436.881,A -85,B 0,C 180,E1 -25339.878,E2 -25339.878} C_VEL
LIN {X 0,Y 130.708,Z 433.214,A -85,B 0,C 180,E1 -25341.066,E2 -25341.066} C_VEL
LIN {X 0,Y 130.241,Z 431.341,A -85,B 0,C 180,E1 -25341.52,E2 -25341.52} C_VEL
LIN {X 0,Y 129.664,Z 428.406,A -85,B 0,C 180,E1 -25347.179,E2 -25347.179} C_VEL
LIN {X 0,Y 129.429,Z 426.601,A -85,B 0,C 180,E1 -25350.881,E2 -25350.881} C_VEL
LIN {X 0,Y 129.041,Z 424.41,A -85,B 0,C 180,E1 -25355.891,E2 -25355.891} C_VEL
LIN {X 0,Y 129.153,Z 424.398,A -85,B 0,C 180,E1 -25360.944,E2 -25360.944} C_VEL
LIN {X 0,Y 129.192,Z 424.392,A -85,B 0,C 180,E1 -25364.298,E2 -25364.298} C_VEL
LIN {X 0,Y 128.505,Z 424.478,A -85,B 0,C 180,E1 -25366.904,E2 -25366.904} C_VEL
LIN {X 0,Y 126.951,Z 424.671,A -85,B 0,C 180,E1 -25369.48,E2 -25369.48} C_VEL
LIN {X 0,Y 123.494,Z 425.094,A -85,B 0,C 180,E1 -25374.763,E2 -25374.763} C_VEL
LIN {X 0,Y 122.739,Z 425.195,A -85,B 0,C 180,E1 -25377.54,E2 -25377.54} C_VEL
LIN {X 0,Y 122.781,Z 425.181,A -85,B 0,C 180,E1 -25378.475,E2 -25378.475} C_VEL
LIN {X 0,Y 123.038,Z 425.157,A -85,B 0,C 180,E1 -25380,E2 -25380} C_VEL
LIN {X 0,Y 122.414,Z 425.229,A -85,B 0,C 180,E1 -25387.171,E2 -25387.171} C_VEL
LIN {X 0,Y 122.36,Z 425.223,A -85,B 0,C 180,E1 -25392.474,E2 -25392.474} C_VEL
LIN {X 0,Y 122.043,Z 425.276,A -85,B 0,C 180,E1 -25400.214,E2 -25400.214} C_VEL
LIN {X 0,Y 121.981,Z 425.272,A -85,B 0,C 180,E1 -25403.786,E2 -25403.786} C_VEL
LIN {X 0,Y 121.94,Z 425.287,A -85,B 0,C 180,E1 -25410.175,E2 -25410.175} C_VEL
LIN {X 0,Y 121.91,Z 425.298,A -85,B 0,C 180,E1 -25416.191,E2 -25416.191} C_VEL
LIN {X 0,Y 121.883,Z 425.287,A -85,B 0,C 180,E1 -25421.446,E2 -25421.446} C_VEL
LIN {X 0,Y 121.871,Z 425.286,A -85,B 0,C 180,E1 -25428.563,E2 -25428.563} C_VEL
LIN {X 0,Y 121.909,Z 425.266,A -85,B 0,C 180,E1 -25434.797,E2 -25434.797} C_VEL
LIN {X 0,Y 121.939,Z 425.299,A -85,B 0,C 180,E1 -25439.83,E2 -25439.83} C_VEL
LIN {X 0,Y 121.984,Z 425.268,A -85,B 0,C 180,E1 -25446.217,E2 -25446.217} C_VEL
LIN {X 0,Y 122.065,Z 425.278,A -85,B 0,C 180,E1 -25448.078,E2 -25448.078} C_VEL
LIN {X 0,Y 122.926,Z 427.92,A -85,B 0,C 180,E1 -25448.878,E2 -25448.878} C_VEL
LIN {X 0,Y 124.846,Z 430.533,A -85,B 0,C 180,E1 -25450.149,E2 -25450.149} C_VEL
LIN {X 0,Y 129.509,Z 438.974,A -85,B 0,C 180,E1 -25453.596,E2 -25453.596} C_VEL
LIN {X 0,Y 133.055,Z 445.925,A -85,B 0,C 180,E1 -25456.331,E2 -25456.331} C_VEL
LIN {X 0,Y 136.319,Z 454.836,A -85,B 0,C 180,E1 -25459.578,E2 -25459.578} C_VEL
LIN {X 0,Y 138.142,Z 466.07,A -85,B 0,C 180,E1 -25463.36,E2 -25463.36} C_VEL
LIN {X 0,Y 138.561,Z 473.469,A -85,B 0,C 180,E1 -25466.002,E2 -25466.002} C_VEL
LIN {X 0,Y 134.748,Z 483.71,A -85,B 0,C 180,E1 -25469.254,E2 -25469.254} C_VEL
LIN {X 0,Y 130.911,Z 492.954,A -85,B 0,C 180,E1 -25473.078,E2 -25473.078} C_VEL
LIN {X 0,Y 127.531,Z 500.796,A -85,B 0,C 180,E1 -25477.273,E2 -25477.273} C_VEL
LIN {X 0,Y 124.443,Z 507.938,A -85,B 0,C 180,E1 -25482.227,E2 -25482.227} C_VEL
LIN {X 0,Y 122.365,Z 512.878,A -85,B 0,C 180,E1 -25486.689,E2 -25486.689} C_VEL
LIN {X 0,Y 120.902,Z 517.03,A -85,B 0,C 180,E1 -25491.552,E2 -25491.552} C_VEL
LIN {X 0,Y 119.921,Z 519.938,A -85,B 0,C 180,E1 -25496.075,E2 -25496.075} C_VEL
LIN {X 0,Y 119.458,Z 522.557,A -85,B 0,C 180,E1 -25501.971,E2 -25501.971} C_VEL
LIN {X 0,Y 119.733,Z 523.617,A -85,B 0,C 180,E1 -25505.943,E2 -25505.943} C_VEL
LIN {X 0,Y 120.735,Z 524.195,A -85,B 0,C 180,E1 -25510.822,E2 -25510.822} C_VEL
LIN {X 0,Y 122.802,Z 523.766,A -85,B 0,C 180,E1 -25516.625,E2 -25516.625} C_VEL
LIN {X 0,Y 125.757,Z 522.2,A -85,B 0,C 180,E1 -25522.066,E2 -25522.066} C_VEL
LIN {X 0,Y 129.543,Z 519.528,A -85,B 0,C 180,E1 -25527.144,E2 -25527.144} C_VEL
LIN {X 0,Y 134.822,Z 515.152,A -85,B 0,C 180,E1 -25532.396,E2 -25532.396} C_VEL
LIN {X 0,Y 141.34,Z 508.839,A -85,B 0,C 180,E1 -25537.389,E2 -25537.389} C_VEL
LIN {X 0,Y 146.796,Z 502.791,A -85,B 0,C 180,E1 -25540.829,E2 -25540.829} C_VEL
LIN {X 0,Y 153.311,Z 494.601,A -85,B 0,C 180,E1 -25544.293,E2 -25544.293} C_VEL
LIN {X 0,Y 154.581,Z 492.647,A -85,B 0,C 180,E1 -25545.037,E2 -25545.037} C_VEL
LIN {X 0,Y 155.629,Z 488.302,A -85,B 0,C 180,E1 -25547.613,E2 -25547.613} C_VEL
LIN {X 0,Y 155.953,Z 485.255,A -85,B 0,C 180,E1 -25549.615,E2 -25549.615} C_VEL
LIN {X 0,Y 155.733,Z 480.651,A -85,B 0,C 180,E1 -25553.128,E2 -25553.128} C_VEL
LIN {X 0,Y 155.095,Z 475.968,A -85,B 0,C 180,E1 -25557.403,E2 -25557.403} C_VEL
LIN {X 0,Y 154.573,Z 473.639,A -85,B 0,C 180,E1 -25560,E2 -25560} C_VEL
LIN {X 0,Y 154.097,Z 471.706,A -85,B 0,C 180,E1 -25562.614,E2 -25562.614} C_VEL
LIN {X 0,Y 153.62,Z 470.151,A -85,B 0,C 180,E1 -25565.25,E2 -25565.25} C_VEL
LIN {X 0,Y 153.146,Z 469.184,A -85,B 0,C 180,E1 -25567.913,E2 -25567.913} C_VEL
LIN {X 0,Y 152.125,Z 469.211,A -85,B 0,C 180,E1 -25574.031,E2 -25574.031} C_VEL
LIN {X 0,Y 152.105,Z 470.356,A -85,B 0,C 180,E1 -25578.871,E2 -25578.871} C_VEL
LIN {X 0,Y 152.585,Z 472.092,A -85,B 0,C 180,E1 -25582.9,E2 -25582.9} C_VEL
LIN {X 0,Y 153.413,Z 476.872,A -85,B 0,C 180,E1 -25588.753,E2 -25588.753} C_VEL
LIN {X 0,Y 154.133,Z 483.152,A -85,B 0,C 180,E1 -25594.034,E2 -25594.034} C_VEL
LIN {X 0,Y 154.571,Z 489.772,A -85,B 0,C 180,E1 -25598.591,E2 -25598.591} C_VEL
LIN {X 0,Y 154.492,Z 491.452,A -85,B 0,C 180,E1 -25599.559,E2 -25599.559} C_VEL
LIN {X 0,Y 151.592,Z 499.72,A -85,B 0,C 180,E1 -25603.191,E2 -25603.191} C_VEL
LIN {X 0,Y 148.171,Z 507.086,A -85,B 0,C 180,E1 -25606.547,E2 -25606.547} C_VEL
LIN {X 0,Y 145.017,Z 512.414,A -85,B 0,C 180,E1 -25609.137,E2 -25609.137} C_VEL
LIN {X 0,Y 139.271,Z 519.272,A -85,B 0,C 180,E1 -25612.731,E2 -25612.731} C_VEL
LIN {X 0,Y 134.052,Z 524.87,A -85,B 0,C 180,E1 -25616.599,E2 -25616.599} C_VEL
LIN {X 0,Y 129.711,Z 529.372,A -85,B 0,C 180,E1 -25620.814,E2 -25620.814} C_VEL
LIN {X 0,Y 125.945,Z 532.869,A -85,B 0,C 180,E1 -25625.259,E2 -25625.259} C_VEL
LIN {X 0,Y 122.957,Z 535.425,A -85,B 0,C 180,E1 -25629.943,E2 -25629.943} C_VEL
LIN {X 0,Y 120.565,Z 537.46,A -85,B 0,C 180,E1 -25636.516,E2 -25636.516} C_VEL
LIN {X 0,Y 119.633,Z 538.007,A -85,B 0,C 180,E1 -25643.252,E2 -25643.252} C_VEL
LIN {X 0,Y 119.682,Z 537.72,A -85,B 0,C 180,E1 -25646.633,E2 -25646.633} C_VEL
LIN {X 0,Y 119.968,Z 537.005,A -85,B 0,C 180,E1 -25649.999,E2 -25649.999} C_VEL
LIN {X 0,Y 119.793,Z 535.484,A -85,B 0,C 180,E1 -25654.172,E2 -25654.172} C_VEL
LIN {X 0,Y 120.109,Z 532.166,A -85,B 0,C 180,E1 -25660.109,E2 -25660.109} C_VEL
LIN {X 0,Y 121.104,Z 528.152,A -85,B 0,C 180,E1 -25665.137,E2 -25665.137} C_VEL
LIN {X 0,Y 123.443,Z 521.964,A -85,B 0,C 180,E1 -25670.843,E2 -25670.843} C_VEL
LIN {X 0,Y 126.266,Z 515.198,A -85,B 0,C 180,E1 -25675.553,E2 -25675.553} C_VEL
LIN {X 0,Y 129.878,Z 506.794,A -85,B 0,C 180,E1 -25680.027,E2 -25680.027} C_VEL
LIN {X 0,Y 132.539,Z 499.954,A -85,B 0,C 180,E1 -25682.922,E2 -25682.922} C_VEL
LIN {X 0,Y 133.843,Z 490.598,A -85,B 0,C 180,E1 -25686.528,E2 -25686.528} C_VEL
LIN {X 0,Y 134.604,Z 479.199,A -85,B 0,C 180,E1 -25690.249,E2 -25690.249} C_VEL
LIN {X 0,Y 134.693,Z 467.57,A -85,B 0,C 180,E1 -25693.506,E2 -25693.506} C_VEL
LIN {X 0,Y 134.228,Z 459.437,A -85,B 0,C 180,E1 -25695.549,E2 -25695.549} C_VEL
LIN {X 0,Y 132.43,Z 452.995,A -85,B 0,C 180,E1 -25697.42,E2 -25697.42} C_VEL
LIN {X 0,Y 129.219,Z 444.69,A -85,B 0,C 180,E1 -25700.025,E2 -25700.025} C_VEL
LIN {X 0,Y 126.754,Z 439.398,A -85,B 0,C 180,E1 -25701.789,E2 -25701.789} C_VEL
LIN {X 0,Y 124.962,Z 435.547,A -85,B 0,C 180,E1 -25703.035,E2 -25703.035} C_VEL
LIN {X 0,Y 123.269,Z 432.351,A -85,B 0,C 180,E1 -25704.167,E2 -25704.167} C_VEL
LIN {X 0,Y 122.905,Z 430.826,A -85,B 0,C 180,E1 -25704.585,E2 -25704.585} C_VEL
LIN {X 0,Y 122.497,Z 428.553,A -85,B 0,C 180,E1 -25709.379,E2 -25709.379} C_VEL
LIN {X 0,Y 122.281,Z 427.075,A -85,B 0,C 180,E1 -25712.627,E2 -25712.627} C_VEL
LIN {X 0,Y 122.052,Z 425.282,A -85,B 0,C 180,E1 -25717.113,E2 -25717.113} C_VEL
LIN {X 0,Y 122.1,Z 425.27,A -85,B 0,C 180,E1 -25724.317,E2 -25724.317} C_VEL
LIN {X 0,Y 122.402,Z 425.238,A -85,B 0,C 180,E1 -25730.082,E2 -25730.082} C_VEL
LIN {X 0,Y 122.781,Z 425.181,A -85,B 0,C 180,E1 -25738.475,E2 -25738.475} C_VEL
LIN {X 0,Y 122.656,Z 425.202,A -85,B 0,C 180,E1 -25740.298,E2 -25740.298} C_VEL
LIN {X 0,Y 121.412,Z 425.355,A -85,B 0,C 180,E1 -25743.004,E2 -25743.004} C_VEL
LIN {X 0,Y 118.043,Z 425.78,A -85,B 0,C 180,E1 -25747.528,E2 -25747.528} C_VEL
LIN {X 0,Y 115.395,Z 426.091,A -85,B 0,C 180,E1 -25752.36,E2 -25752.36} C_VEL
LIN {X 0,Y 115.21,Z 426.113,A -85,B 0,C 180,E1 -25753.367,E2 -25753.367} C_VEL
LIN {X 0,Y 115.01,Z 426.159,A -85,B 0,C 180,E1 -25757.791,E2 -25757.791} C_VEL
LIN {X 0,Y 114.944,Z 426.147,A -85,B 0,C 180,E1 -25763.493,E2 -25763.493} C_VEL
LIN {X 0,Y 114.867,Z 426.162,A -85,B 0,C 180,E1 -25771.069,E2 -25771.069} C_VEL
LIN {X 0,Y 114.801,Z 426.184,A -85,B 0,C 180,E1 -25777.749,E2 -25777.749} C_VEL
LIN {X 0,Y 114.793,Z 426.175,A -85,B 0,C 180,E1 -25782.722,E2 -25782.722} C_VEL
LIN {X 0,Y 114.793,Z 426.176,A -85,B 0,C 180,E1 -25787.668,E2 -25787.668} C_VEL
LIN {X 0,Y 114.786,Z 426.138,A -85,B 0,C 180,E1 -25792.746,E2 -25792.746} C_VEL
LIN {X 0,Y 114.861,Z 426.183,A -85,B 0,C 180,E1 -25798.94,E2 -25798.94} C_VEL
LIN {X 0,Y 114.876,Z 426.202,A -85,B 0,C 180,E1 -25804.645,E2 -25804.645} C_VEL
LIN {X 0,Y 115.776,Z 428.79,A -85,B 0,C 180,E1 -25805.583,E2 -25805.583} C_VEL
LIN {X 0,Y 117.813,Z 431.417,A -85,B 0,C 180,E1 -25807.108,E2 -25807.108} C_VEL
LIN {X 0,Y 119.625,Z 434.549,A -85,B 0,C 180,E1 -25808.592,E2 -25808.592} C_VEL
LIN {X 0,Y 124.101,Z 442.645,A -85,B 0,C 180,E1 -25812.28,E2 -25812.28} C_VEL
LIN {X 0,Y 127.918,Z 450.763,A -85,B 0,C 180,E1 -25815.771,E2 -25815.771} C_VEL
LIN {X 0,Y 130.441,Z 458.275,A -85,B 0,C 180,E1 -25818.716,E2 -25818.716} C_VEL
LIN {X 0,Y 131.817,Z 468.49,A -85,B 0,C 180,E1 -25822.467,E2 -25822.467} C_VEL
LIN {X 0,Y 132.068,Z 474.215,A -85,B 0,C 180,E1 -25824.657,E2 -25824.657} C_VEL
LIN {X 0,Y 128.243,Z 484.323,A -85,B 0,C 180,E1 -25828.038,E2 -25828.038} C_VEL
LIN {X 0,Y 124.607,Z 492.709,A -85,B 0,C 180,E1 -25831.617,E2 -25831.617} C_VEL
LIN {X 0,Y 121.093,Z 500.417,A -85,B 0,C 180,E1 -25835.83,E2 -25835.83} C_VEL
LIN {X 0,Y 117.686,Z 507.913,A -85,B 0,C 180,E1 -25841.192,E2 -25841.192} C_VEL
LIN {X 0,Y 115.433,Z 513.014,A -85,B 0,C 180,E1 -25845.969,E2 -25845.969} C_VEL
LIN {X 0,Y 113.644,Z 517.822,A -85,B 0,C 180,E1 -25851.929,E2 -25851.929} C_VEL
LIN {X 0,Y 112.469,Z 521.666,A -85,B 0,C 180,E1 -25858.973,E2 -25858.973} C_VEL
LIN {X 0,Y 112.636,Z 523.877,A -85,B 0,C 180,E1 -25865.791,E2 -25865.791} C_VEL
LIN {X 0,Y 114.117,Z 524.645,A -85,B 0,C 180,E1 -25872.644,E2 -25872.644} C_VEL
LIN {X 0,Y 116.402,Z 524.164,A -85,B 0,C 180,E1 -25878.382,E2 -25878.382} C_VEL
LIN {X 0,Y 120.288,Z 522.215,A -85,B 0,C 180,E1 -25884.882,E2 -25884.882} C_VEL
LIN {X 0,Y 125.25,Z 518.884,A -85,B 0,C 180,E1 -25890.707,E2 -25890.707} C_VEL
LIN {X 0,Y 131.014,Z 514.246,A -85,B 0,C 180,E1 -25895.773,E2 -25895.773} C_VEL
LIN {X 0,Y 136.703,Z 509.01,A -85,B 0,C 180,E1 -25899.758,E2 -25899.758} C_VEL
LIN {X 0,Y 143.352,Z 502.025,A -85,B 0,C 180,E1 -25903.612,E2 -25903.612} C_VEL
LIN {X 0,Y 148.671,Z 495.565,A -85,B 0,C 180,E1 -25906.328,E2 -25906.328} C_VEL
LIN {X 0,Y 149.465,Z 494.005,A -85,B 0,C 180,E1 -25907.163,E2 -25907.163} C_VEL
LIN {X 0,Y 150.286,Z 490.954,A -85,B 0,C 180,E1 -25909.219,E2 -25909.219} C_VEL
LIN {X 0,Y 150.648,Z 487.396,A -85,B 0,C 180,E1 -25911.954,E2 -25911.954} C_VEL
LIN {X 0,Y 150.567,Z 482.956,A -85,B 0,C 180,E1 -25915.985,E2 -25915.985} C_VEL
LIN {X 0,Y 150.187,Z 479.374,A -85,B 0,C 180,E1 -25920,E2 -25920} C_VEL
LIN {X 0,Y 149.86,Z 477.482,A -85,B 0,C 180,E1 -25922.688,E2 -25922.688} C_VEL
LIN {X 0,Y 149.556,Z 476.003,A -85,B 0,C 180,E1 -25925.393,E2 -25925.393} C_VEL
LIN {X 0,Y 149.136,Z 475.062,A -85,B 0,C 180,E1 -25928.265,E2 -25928.265} C_VEL
LIN {X 0,Y 148.309,Z 475.123,A -85,B 0,C 180,E1 -25933.706,E2 -25933.706} C_VEL
LIN {X 0,Y 148.212,Z 476.522,A -85,B 0,C 180,E1 -25939.386,E2 -25939.386} C_VEL
LIN {X 0,Y 148.501,Z 477.715,A -85,B 0,C 180,E1 -25942.247,E2 -25942.247} C_VEL
LIN {X 0,Y 148.968,Z 482.169,A -85,B 0,C 180,E1 -25948.15,E2 -25948.15} C_VEL
LIN {X 0,Y 149.191,Z 487.274,A -85,B 0,C 180,E1 -25952.8,E2 -25952.8} C_VEL
LIN {X 0,Y 149.184,Z 493.862,A -85,B 0,C 180,E1 -25957.765,E2 -25957.765} C_VEL
LIN {X 0,Y 148.565,Z 496.203,A -85,B 0,C 180,E1 -25959.005,E2 -25959.005} C_VEL
LIN {X 0,Y 145.04,Z 504.046,A -85,B 0,C 180,E1 -25962.717,E2 -25962.717} C_VEL
LIN {X 0,Y 141.365,Z 510.369,A -85,B 0,C 180,E1 -25965.892,E2 -25965.892} C_VEL
LIN {X 0,Y 138.751,Z 514.081,A -85,B 0,C 180,E1 -25967.845,E2 -25967.845} C_VEL
LIN {X 0,Y 131.762,Z 521.531,A -85,B 0,C 180,E1 -25972.165,E2 -25972.165} C_VEL
LIN {X 0,Y 125.86,Z 527.222,A -85,B 0,C 180,E1 -25976.887,E2 -25976.887} C_VEL
LIN {X 0,Y 120.715,Z 531.711,A -85,B 0,C 180,E1 -25982.24,E2 -25982.24} C_VEL
LIN {X 0,Y 118.359,Z 533.663,A -85,B 0,C 180,E1 -25985.439,E2 -25985.439} C_VEL
LIN {X 0,Y 116.292,Z 535.191,A -85,B 0,C 180,E1 -25988.739,E2 -25988.739} C_VEL
LIN {X 0,Y 113.642,Z 537.101,A -85,B 0,C 180,E1 -25995.677,E2 -25995.677} C_VEL
LIN {X 0,Y 112.571,Z 537.541,A -85,B 0,C 180,E1 -26002.826,E2 -26002.826} C_VEL
LIN {X 0,Y 112.621,Z 537.093,A -85,B 0,C 180,E1 -26006.821,E2 -26006.821} C_VEL
LIN {X 0,Y 112.904,Z 536.399,A -85,B 0,C 180,E1 -26009.999,E2 -26009.999} C_VEL
LIN {X 0,Y 112.719,Z 535.007,A -85,B 0,C 180,E1 -26013.976,E2 -26013.976} C_VEL
LIN {X 0,Y 112.869,Z 532.468,A -85,B 0,C 180,E1 -26018.954,E2 -26018.954} C_VEL
LIN {X 0,Y 113.778,Z 528.718,A -85,B 0,C 180,E1 -26024.303,E2 -26024.303} C_VEL
LIN {X 0,Y 115.523,Z 523.818,A -85,B 0,C 180,E1 -26029.547,E2 -26029.547} C_VEL
LIN {X 0,Y 118.223,Z 517.644,A -85,B 0,C 180,E1 -26034.589,E2 -26034.589} C_VEL
LIN {X 0,Y 121.551,Z 510.141,A -85,B 0,C 180,E1 -26039.286,E2 -26039.286} C_VEL
LIN {X 0,Y 125.192,Z 502.018,A -85,B 0,C 180,E1 -26043.182,E2 -26043.182} C_VEL
LIN {X 0,Y 126.385,Z 497.243,A -85,B 0,C 180,E1 -26045.233,E2 -26045.233} C_VEL
LIN {X 0,Y 127.608,Z 487.399,A -85,B 0,C 180,E1 -26049.077,E2 -26049.077} C_VEL
LIN {X 0,Y 128.412,Z 476.073,A -85,B 0,C 180,E1 -26052.809,E2 -26052.809} C_VEL
LIN {X 0,Y 128.37,Z 464.716,A -85,B 0,C 180,E1 -26056.061,E2 -26056.061} C_VEL
LIN {X 0,Y 127.83,Z 459.837,A -85,B 0,C 180,E1 -26057.449,E2 -26057.449} C_VEL
LIN {X 0,Y 124.702,Z 450.376,A -85,B 0,C 180,E1 -26060.652,E2 -26060.652} C_VEL
LIN {X 0,Y 121.242,Z 442.349,A -85,B 0,C 180,E1 -26063.548,E2 -26063.548} C_VEL
LIN {X 0,Y 119.997,Z 439.716,A -85,B 0,C 180,E1 -26064.536,E2 -26064.536} C_VEL
LIN {X 0,Y 117.943,Z 435.42,A -85,B 0,C 180,E1 -26066.167,E2 -26066.167} C_VEL
LIN {X 0,Y 116.007,Z 432.118,A -85,B 0,C 180,E1 -26067.632,E2 -26067.632} C_VEL
LIN {X 0,Y 115.557,Z 430.319,A -85,B 0,C 180,E1 -26068.14,E2 -26068.14} C_VEL
LIN {X 0,Y 115.125,Z 427.528,A -85,B 0,C 180,E1 -26074.702,E2 -26074.702} C_VEL
LIN {X 0,Y 114.992,Z 426.161,A -85,B 0,C 180,E1 -26078.488,E2 -26078.488} C_VEL
LIN {X 0,Y 115.131,Z 426.144,A -85,B 0,C 180,E1 -26085.867,E2 -26085.867} C_VEL
LIN {X 0,Y 115.321,Z 426.12,A -85,B 0,C 180,E1 -26089.466,E2 -26089.466} C_VEL
LIN {X 0,Y 115.517,Z 426.088,A -85,B 0,C 180,E1 -26096.512,E2 -26096.512} C_VEL
LIN {X 0,Y 115.99,Z 426.034,A -85,B 0,C 180,E1 -26100,E2 -26100} C_VEL
LIN {X 0,Y 115.381,Z 426.11,A -85,B 0,C 180,E1 -26107.062,E2 -26107.062} C_VEL
LIN {X 0,Y 115.281,Z 426.104,A -85,B 0,C 180,E1 -26112.739,E2 -26112.739} C_VEL
LIN {X 0,Y 115.21,Z 426.113,A -85,B 0,C 180,E1 -26113.367,E2 -26113.367} C_VEL
LIN {X 0,Y 114.306,Z 426.242,A -85,B 0,C 180,E1 -26116.281,E2 -26116.281} C_VEL
LIN {X 0,Y 112.59,Z 426.459,A -85,B 0,C 180,E1 -26119.158,E2 -26119.158} C_VEL
LIN {X 0,Y 107.995,Z 427.032,A -85,B 0,C 180,E1 -26127.175,E2 -26127.175} C_VEL
LIN {X 0,Y 107.706,Z 427.05,A -85,B 0,C 180,E1 -26129.307,E2 -26129.307} C_VEL
LIN {X 0,Y 107.792,Z 427.039,A -85,B 0,C 180,E1 -26132.053,E2 -26132.053} C_VEL
LIN {X 0,Y 107.706,Z 427.065,A -85,B 0,C 180,E1 -26138.465,E2 -26138.465} C_VEL
LIN {X 0,Y 107.678,Z 427.073,A -85,B 0,C 180,E1 -26145.887,E2 -26145.887} C_VEL
LIN {X 0,Y 107.685,Z 427.021,A -85,B 0,C 180,E1 -26151.553,E2 -26151.553} C_VEL
LIN {X 0,Y 107.796,Z 427.064,A -85,B 0,C 180,E1 -26158.564,E2 -26158.564} C_VEL
LIN {X 0,Y 107.845,Z 427.048,A -85,B 0,C 180,E1 -26160.593,E2 -26160.593} C_VEL
LIN {X 0,Y 108.672,Z 429.62,A -85,B 0,C 180,E1 -26161.687,E2 -26161.687} C_VEL
LIN {X 0,Y 110.758,Z 432.16,A -85,B 0,C 180,E1 -26163.466,E2 -26163.466} C_VEL
LIN {X 0,Y 112.629,Z 435.461,A -85,B 0,C 180,E1 -26165.265,E2 -26165.265} C_VEL
LIN {X 0,Y 116.959,Z 442.924,A -85,B 0,C 180,E1 -26169.259,E2 -26169.259} C_VEL
LIN {X 0,Y 121.4,Z 452.299,A -85,B 0,C 180,E1 -26173.746,E2 -26173.746} C_VEL
LIN {X 0,Y 123.863,Z 459.413,A -85,B 0,C 180,E1 -26176.883,E2 -26176.883} C_VEL
LIN {X 0,Y 124.802,Z 464.219,A -85,B 0,C 180,E1 -26178.825,E2 -26178.825} C_VEL
LIN {X 0,Y 125.565,Z 472.038,A -85,B 0,C 180,E1 -26181.957,E2 -26181.957} C_VEL
LIN {X 0,Y 125.467,Z 476.05,A -85,B 0,C 180,E1 -26183.569,E2 -26183.569} C_VEL
LIN {X 0,Y 121.101,Z 486.504,A -85,B 0,C 180,E1 -26187.352,E2 -26187.352} C_VEL
LIN {X 0,Y 116.785,Z 495.737,A -85,B 0,C 180,E1 -26191.725,E2 -26191.725} C_VEL
LIN {X 0,Y 113.168,Z 503.321,A -85,B 0,C 180,E1 -26196.459,E2 -26196.459} C_VEL
LIN {X 0,Y 110.433,Z 508.992,A -85,B 0,C 180,E1 -26201.007,E2 -26201.007} C_VEL
LIN {X 0,Y 107.898,Z 514.73,A -85,B 0,C 180,E1 -26207.045,E2 -26207.045} C_VEL
LIN {X 0,Y 106.193,Z 519.152,A -85,B 0,C 180,E1 -26213.397,E2 -26213.397} C_VEL
LIN {X 0,Y 105.335,Z 522.286,A -85,B 0,C 180,E1 -26219.845,E2 -26219.845} C_VEL
LIN {X 0,Y 105.689,Z 524.409,A -85,B 0,C 180,E1 -26227.063,E2 -26227.063} C_VEL
LIN {X 0,Y 107.338,Z 525.102,A -85,B 0,C 180,E1 -26233.926,E2 -26233.926} C_VEL
LIN {X 0,Y 110.085,Z 524.575,A -85,B 0,C 180,E1 -26240.325,E2 -26240.325} C_VEL
LIN {X 0,Y 113.792,Z 522.931,A -85,B 0,C 180,E1 -26246.23,E2 -26246.23} C_VEL
LIN {X 0,Y 119.078,Z 519.777,A -85,B 0,C 180,E1 -26252.289,E2 -26252.289} C_VEL
LIN {X 0,Y 125.668,Z 514.936,A -85,B 0,C 180,E1 -26257.851,E2 -26257.851} C_VEL
LIN {X 0,Y 132.657,Z 508.914,A -85,B 0,C 180,E1 -26262.48,E2 -26262.48} C_VEL
LIN {X 0,Y 139.359,Z 502.225,A -85,B 0,C 180,E1 -26266.118,E2 -26266.118} C_VEL
LIN {X 0,Y 143.597,Z 497.357,A -85,B 0,C 180,E1 -26268.193,E2 -26268.193} C_VEL
LIN {X 0,Y 144.791,Z 494.021,A -85,B 0,C 180,E1 -26270.609,E2 -26270.609} C_VEL
LIN {X 0,Y 145.305,Z 491.206,A -85,B 0,C 180,E1 -26273.055,E2 -26273.055} C_VEL
LIN {X 0,Y 145.499,Z 487.106,A -85,B 0,C 180,E1 -26277.231,E2 -26277.231} C_VEL
LIN {X 0,Y 145.494,Z 484.888,A -85,B 0,C 180,E1 -26280,E2 -26280} C_VEL
LIN {X 0,Y 145.309,Z 483.044,A -85,B 0,C 180,E1 -26282.772,E2 -26282.772} C_VEL
LIN {X 0,Y 145.204,Z 481.62,A -85,B 0,C 180,E1 -26285.555,E2 -26285.555} C_VEL
LIN {X 0,Y 144.894,Z 480.761,A -85,B 0,C 180,E1 -26288.367,E2 -26288.367} C_VEL
LIN {X 0,Y 144.083,Z 480.959,A -85,B 0,C 180,E1 -26294.116,E2 -26294.116} C_VEL
LIN {X 0,Y 143.972,Z 481.562,A -85,B 0,C 180,E1 -26297.031,E2 -26297.031} C_VEL
LIN {X 0,Y 144.17,Z 483.44,A -85,B 0,C 180,E1 -26302.149,E2 -26302.149} C_VEL
LIN {X 0,Y 144.264,Z 487.308,A -85,B 0,C 180,E1 -26307.57,E2 -26307.57} C_VEL
LIN {X 0,Y 144.087,Z 492.31,A -85,B 0,C 180,E1 -26312.448,E2 -26312.448} C_VEL
LIN {X 0,Y 143.695,Z 497.666,A -85,B 0,C 180,E1 -26316.808,E2 -26316.808} C_VEL
LIN {X 0,Y 141.231,Z 502.905,A -85,B 0,C 180,E1 -26319.53,E2 -26319.53} C_VEL
LIN {X 0,Y 137.095,Z 509.812,A -85,B 0,C 180,E1 -26323.154,E2 -26323.154} C_VEL
LIN {X 0,Y 133.555,Z 514.576,A -85,B 0,C 180,E1 -26325.793,E2 -26325.793} C_VEL
LIN {X 0,Y 128.287,Z 519.871,A -85,B 0,C 180,E1 -26328.898,E2 -26328.898} C_VEL
LIN {X 0,Y 122.41,Z 525.166,A -85,B 0,C 180,E1 -26332.926,E2 -26332.926} C_VEL
LIN {X 0,Y 117.463,Z 529.378,A -85,B 0,C 180,E1 -26337.419,E2 -26337.419} C_VEL
LIN {X 0,Y 114.466,Z 531.661,A -85,B 0,C 180,E1 -26340.581,E2 -26340.581} C_VEL
LIN {X 0,Y 111.923,Z 533.506,A -85,B 0,C 180,E1 -26343.924,E2 -26343.924} C_VEL
LIN {X 0,Y 107.943,Z 536.025,A -85,B 0,C 180,E1 -26351.001,E2 -26351.001} C_VEL
LIN {X 0,Y 105.924,Z 537.091,A -85,B 0,C 180,E1 -26358.518,E2 -26358.518} C_VEL
LIN {X 0,Y 105.528,Z 536.595,A -85,B 0,C 180,E1 -26366.18,E2 -26366.18} C_VEL
LIN {X 0,Y 105.839,Z 535.775,A -85,B 0,C 180,E1 -26369.999,E2 -26369.999} C_VEL
LIN {X 0,Y 105.654,Z 534.487,A -85,B 0,C 180,E1 -26373.813,E2 -26373.813} C_VEL
LIN {X 0,Y 105.857,Z 531.679,A -85,B 0,C 180,E1 -26379.553,E2 -26379.553} C_VEL
LIN {X 0,Y 106.872,Z 527.809,A -85,B 0,C 180,E1 -26385.249,E2 -26385.249} C_VEL
LIN {X 0,Y 108.823,Z 522.789,A -85,B 0,C 180,E1 -26390.804,E2 -26390.804} C_VEL
LIN {X 0,Y 111.774,Z 516.466,A -85,B 0,C 180,E1 -26396.111,E2 -26396.111} C_VEL
LIN {X 0,Y 115.223,Z 509.065,A -85,B 0,C 180,E1 -26400.846,E2 -26400.846} C_VEL
LIN {X 0,Y 118.467,Z 502.211,A -85,B 0,C 180,E1 -26404.3,E2 -26404.3} C_VEL
LIN {X 0,Y 119.572,Z 498.51,A -85,B 0,C 180,E1 -26405.996,E2 -26405.996} C_VEL
LIN {X 0,Y 121.023,Z 488.6,A -85,B 0,C 180,E1 -26410.167,E2 -26410.167} C_VEL
LIN {X 0,Y 121.996,Z 478.644,A -85,B 0,C 180,E1 -26413.731,E2 -26413.731} C_VEL
LIN {X 0,Y 122.332,Z 468.46,A -85,B 0,C 180,E1 -26416.95,E2 -26416.95} C_VEL
LIN {X 0,Y 122.141,Z 463.601,A -85,B 0,C 180,E1 -26418.416,E2 -26418.416} C_VEL
LIN {X 0,Y 119.405,Z 454.378,A -85,B 0,C 180,E1 -26421.829,E2 -26421.829} C_VEL
LIN {X 0,Y 115.145,Z 443.957,A -85,B 0,C 180,E1 -26426.023,E2 -26426.023} C_VEL
LIN {X 0,Y 113.269,Z 439.934,A -85,B 0,C 180,E1 -26427.758,E2 -26427.758} C_VEL
LIN {X 0,Y 111.333,Z 435.934,A -85,B 0,C 180,E1 -26429.518,E2 -26429.518} C_VEL
LIN {X 0,Y 108.633,Z 431.216,A -85,B 0,C 180,E1 -26431.897,E2 -26431.897} C_VEL
LIN {X 0,Y 108.235,Z 429.709,A -85,B 0,C 180,E1 -26432.442,E2 -26432.442} C_VEL
LIN {X 0,Y 107.958,Z 427.218,A -85,B 0,C 180,E1 -26439.02,E2 -26439.02} C_VEL
LIN {X 0,Y 108.169,Z 427.011,A -85,B 0,C 180,E1 -26447.045,E2 -26447.045} C_VEL
LIN {X 0,Y 108.3,Z 426.984,A -85,B 0,C 180,E1 -26452.543,E2 -26452.543} C_VEL
LIN {X 0,Y 108.939,Z 426.912,A -85,B 0,C 180,E1 -26460,E2 -26460} C_VEL
LIN {X 0,Y 108.326,Z 426.991,A -85,B 0,C 180,E1 -26467.456,E2 -26467.456} C_VEL
LIN {X 0,Y 108.18,Z 426.987,A -85,B 0,C 180,E1 -26473.164,E2 -26473.164} C_VEL
LIN {X 0,Y 107.902,Z 427.043,A -85,B 0,C 180,E1 -26479.006,E2 -26479.006} C_VEL
LIN {X 0,Y 107.855,Z 427.032,A -85,B 0,C 180,E1 -26484.185,E2 -26484.185} C_VEL
LIN {X 0,Y 107.706,Z 427.05,A -85,B 0,C 180,E1 -26489.307,E2 -26489.307} C_VEL
LIN {X 0,Y 107.086,Z 427.13,A -85,B 0,C 180,E1 -26492.432,E2 -26492.432} C_VEL
LIN {X 0,Y 105.564,Z 427.338,A -85,B 0,C 180,E1 -26495.525,E2 -26495.525} C_VEL
LIN {X 0,Y 101.005,Z 427.92,A -85,B 0,C 180,E1 -26504.136,E2 -26504.136} C_VEL
LIN {X 0,Y 100.606,Z 427.942,A -85,B 0,C 180,E1 -26506.429,E2 -26506.429} C_VEL
LIN {X 0,Y 100.624,Z 427.901,A -85,B 0,C 180,E1 -26511.055,E2 -26511.055} C_VEL
LIN {X 0,Y 100.659,Z 427.988,A -85,B 0,C 180,E1 -26515.593,E2 -26515.593} C_VEL
LIN {X 0,Y 101.509,Z 430.465,A -85,B 0,C 180,E1 -26516.859,E2 -26516.859} C_VEL
LIN {X 0,Y 104.031,Z 433.42,A -85,B 0,C 180,E1 -26519.469,E2 -26519.469} C_VEL
LIN {X 0,Y 105.896,Z 436.643,A -85,B 0,C 180,E1 -26521.581,E2 -26521.581} C_VEL
LIN {X 0,Y 106.864,Z 438.192,A -85,B 0,C 180,E1 -26522.591,E2 -26522.591} C_VEL
LIN {X 0,Y 110.285,Z 444.206,A -85,B 0,C 180,E1 -26526.239,E2 -26526.239} C_VEL
LIN {X 0,Y 113.813,Z 451.473,A -85,B 0,C 180,E1 -26530.254,E2 -26530.254} C_VEL
LIN {X 0,Y 116.929,Z 459.004,A -85,B 0,C 180,E1 -26534.089,E2 -26534.089} C_VEL
LIN {X 0,Y 118.522,Z 465.229,A -85,B 0,C 180,E1 -26536.999,E2 -26536.999} C_VEL
LIN {X 0,Y 119.204,Z 473.677,A -85,B 0,C 180,E1 -26540.67,E2 -26540.67} C_VEL
LIN {X 0,Y 119.19,Z 476.609,A -85,B 0,C 180,E1 -26541.951,E2 -26541.951} C_VEL
LIN {X 0,Y 114.983,Z 486.386,A -85,B 0,C 180,E1 -26545.619,E2 -26545.619} C_VEL
LIN {X 0,Y 110.561,Z 495.405,A -85,B 0,C 180,E1 -26550.001,E2 -26550.001} C_VEL
LIN {X 0,Y 106.739,Z 502.976,A -85,B 0,C 180,E1 -26554.84,E2 -26554.84} C_VEL
LIN {X 0,Y 103.21,Z 509.991,A -85,B 0,C 180,E1 -26560.794,E2 -26560.794} C_VEL
LIN {X 0,Y 100.972,Z 514.798,A -85,B 0,C 180,E1 -26566.166,E2 -26566.166} C_VEL
LIN {X 0,Y 99.157,Z 519.267,A -85,B 0,C 180,E1 -26572.865,E2 -26572.865} C_VEL
LIN {X 0,Y 98.196,Z 522.891,A -85,B 0,C 180,E1 -26580.81,E2 -26580.81} C_VEL
LIN {X 0,Y 98.819,Z 524.92,A -85,B 0,C 180,E1 -26588.526,E2 -26588.526} C_VEL
LIN {X 0,Y 100.777,Z 525.557,A -85,B 0,C 180,E1 -26595.782,E2 -26595.782} C_VEL
LIN {X 0,Y 104.612,Z 524.778,A -85,B 0,C 180,E1 -26603.724,E2 -26603.724} C_VEL
LIN {X 0,Y 108.084,Z 523.308,A -85,B 0,C 180,E1 -26608.654,E2 -26608.654} C_VEL
LIN {X 0,Y 113.203,Z 520.525,A -85,B 0,C 180,E1 -26614.241,E2 -26614.241} C_VEL
LIN {X 0,Y 119.905,Z 516.13,A -85,B 0,C 180,E1 -26619.686,E2 -26619.686} C_VEL
LIN {X 0,Y 126.291,Z 511.133,A -85,B 0,C 180,E1 -26623.844,E2 -26623.844} C_VEL
LIN {X 0,Y 133.825,Z 504.248,A -85,B 0,C 180,E1 -26627.873,E2 -26627.873} C_VEL
LIN {X 0,Y 138.525,Z 499.284,A -85,B 0,C 180,E1 -26630.194,E2 -26630.194} C_VEL
LIN {X 0,Y 139.589,Z 496.355,A -85,B 0,C 180,E1 -26632.769,E2 -26632.769} C_VEL
LIN {X 0,Y 140.271,Z 492.32,A -85,B 0,C 180,E1 -26637.128,E2 -26637.128} C_VEL
LIN {X 0,Y 140.485,Z 490.124,A -85,B 0,C 180,E1 -26640,E2 -26640} C_VEL
LIN {X 0,Y 140.493,Z 488.358,A -85,B 0,C 180,E1 -26642.867,E2 -26642.867} C_VEL
LIN {X 0,Y 140.55,Z 486.966,A -85,B 0,C 180,E1 -26645.739,E2 -26645.739} C_VEL
LIN {X 0,Y 140.314,Z 486.246,A -85,B 0,C 180,E1 -26648.642,E2 -26648.642} C_VEL
LIN {X 0,Y 139.564,Z 486.583,A -85,B 0,C 180,E1 -26654.583,E2 -26654.583} C_VEL
LIN {X 0,Y 139.455,Z 487.269,A -85,B 0,C 180,E1 -26657.6,E2 -26657.6} C_VEL
LIN {X 0,Y 139.48,Z 488.292,A -85,B 0,C 180,E1 -26660.653,E2 -26660.653} C_VEL
LIN {X 0,Y 139.285,Z 490.709,A -85,B 0,C 180,E1 -26664.738,E2 -26664.738} C_VEL
LIN {X 0,Y 139.33,Z 492.229,A -85,B 0,C 180,E1 -26666.999,E2 -26666.999} C_VEL
LIN {X 0,Y 138.729,Z 497.161,A -85,B 0,C 180,E1 -26672.134,E2 -26672.134} C_VEL
LIN {X 0,Y 138.176,Z 500.966,A -85,B 0,C 180,E1 -26675.532,E2 -26675.532} C_VEL
LIN {X 0,Y 134.847,Z 506.683,A -85,B 0,C 180,E1 -26678.713,E2 -26678.713} C_VEL
LIN {X 0,Y 130.454,Z 512.748,A -85,B 0,C 180,E1 -26682.204,E2 -26682.204} C_VEL
LIN {X 0,Y 127.473,Z 516.128,A -85,B 0,C 180,E1 -26684.215,E2 -26684.215} C_VEL
LIN {X 0,Y 120.876,Z 522.032,A -85,B 0,C 180,E1 -26688.038,E2 -26688.038} C_VEL
LIN {X 0,Y 114.942,Z 526.785,A -85,B 0,C 180,E1 -26692.306,E2 -26692.306} C_VEL
LIN {X 0,Y 109.916,Z 530.516,A -85,B 0,C 180,E1 -26697.078,E2 -26697.078} C_VEL
LIN {X 0,Y 105.549,Z 533.332,A -85,B 0,C 180,E1 -26702.218,E2 -26702.218} C_VEL
LIN {X 0,Y 101.216,Z 535.732,A -85,B 0,C 180,E1 -26709.684,E2 -26709.684} C_VEL
LIN {X 0,Y 99.868,Z 536.383,A -85,B 0,C 180,E1 -26713.65,E2 -26713.65} C_VEL
LIN {X 0,Y 98.479,Z 536.512,A -85,B 0,C 180,E1 -26721.793,E2 -26721.793} C_VEL
LIN {X 0,Y 98.511,Z 535.816,A -85,B 0,C 180,E1 -26727.185,E2 -26727.185} C_VEL
LIN {X 0,Y 98.776,Z 535.154,A -85,B 0,C 180,E1 -26729.999,E2 -26729.999} C_VEL
LIN {X 0,Y 98.56,Z 533.783,A -85,B 0,C 180,E1 -26734.088,E2 -26734.088} C_VEL
LIN {X 0,Y 98.85,Z 530.874,A -85,B 0,C 180,E1 -26740.237,E2 -26740.237} C_VEL
LIN {X 0,Y 100.015,Z 526.881,A -85,B 0,C 180,E1 -26746.323,E2 -26746.323} C_VEL
LIN {X 0,Y 102.685,Z 520.708,A -85,B 0,C 180,E1 -26753.174,E2 -26753.174} C_VEL
LIN {X 0,Y 106.018,Z 513.965,A -85,B 0,C 180,E1 -26758.723,E2 -26758.723} C_VEL
LIN {X 0,Y 109.697,Z 506.586,A -85,B 0,C 180,E1 -26763.356,E2 -26763.356} C_VEL
LIN {X 0,Y 112.52,Z 500.538,A -85,B 0,C 180,E1 -26766.394,E2 -26766.394} C_VEL
LIN {X 0,Y 114.317,Z 491.117,A -85,B 0,C 180,E1 -26770.782,E2 -26770.782} C_VEL
LIN {X 0,Y 115.649,Z 480.61,A -85,B 0,C 180,E1 -26774.943,E2 -26774.943} C_VEL
LIN {X 0,Y 116.256,Z 470.784,A -85,B 0,C 180,E1 -26778.319,E2 -26778.319} C_VEL
LIN {X 0,Y 116.309,Z 467.093,A -85,B 0,C 180,E1 -26779.491,E2 -26779.491} C_VEL
LIN {X 0,Y 114.214,Z 458.81,A -85,B 0,C 180,E1 -26782.828,E2 -26782.828} C_VEL
LIN {X 0,Y 110.517,Z 448.714,A -85,B 0,C 180,E1 -26787.28,E2 -26787.28} C_VEL
LIN {X 0,Y 108.661,Z 444.583,A -85,B 0,C 180,E1 -26789.246,E2 -26789.246} C_VEL
LIN {X 0,Y 106.407,Z 439.775,A -85,B 0,C 180,E1 -26791.659,E2 -26791.659} C_VEL
LIN {X 0,Y 104.317,Z 435.287,A -85,B 0,C 180,E1 -26793.987,E2 -26793.987} C_VEL
LIN {X 0,Y 101.954,Z 431.808,A -85,B 0,C 180,E1 -26796.38,E2 -26796.38} C_VEL
LIN {X 0,Y 101.063,Z 429.06,A -85,B 0,C 180,E1 -26797.648,E2 -26797.648} C_VEL
LIN {X 0,Y 100.873,Z 427.92,A -85,B 0,C 180,E1 -26801.729,E2 -26801.729} C_VEL
LIN {X 0,Y 101.153,Z 427.885,A -85,B 0,C 180,E1 -26807.97,E2 -26807.97} C_VEL
LIN {X 0,Y 101.238,Z 427.866,A -85,B 0,C 180,E1 -26812.02,E2 -26812.02} C_VEL
LIN {X 0,Y 101.863,Z 427.793,A -85,B 0,C 180,E1 -26820,E2 -26820} C_VEL
LIN {X 0,Y 101.265,Z 427.871,A -85,B 0,C 180,E1 -26827.979,E2 -26827.979} C_VEL
LIN {X 0,Y 101.122,Z 427.866,A -85,B 0,C 180,E1 -26833.353,E2 -26833.353} C_VEL
LIN {X 0,Y 100.813,Z 427.917,A -85,B 0,C 180,E1 -26840.4,E2 -26840.4} C_VEL
LIN {X 0,Y 100.772,Z 427.918,A -85,B 0,C 180,E1 -26844.96,E2 -26844.96} C_VEL
LIN {X 0,Y 100.698,Z 427.922,A -85,B 0,C 180,E1 -26853.125,E2 -26853.125} C_VEL
LIN {X 0,Y 100.653,Z 427.933,A -85,B 0,C 180,E1 -26859.823,E2 -26859.823} C_VEL
LIN {X 0,Y 100.606,Z 427.942,A -85,B 0,C 180,E1 -26866.429,E2 -26866.429} C_VEL
LIN {X 0,Y 100.484,Z 428.383,A -85,B 0,C 180,E1 -26868.638,E2 -26868.638} C_VEL
LIN {X 0,Y 100.351,Z 430.405,A -85,B 0,C 180,E1 -26871.796,E2 -26871.796} C_VEL
LIN {X 0,Y 100.412,Z 433.502,A -85,B 0,C 180,E1 -26874.696,E2 -26874.696} C_VEL
LIN {X 0,Y 101.069,Z 438.662,A -85,B 0,C 180,E1 -26878.336,E2 -26878.336} C_VEL
LIN {X 0,Y 102.856,Z 443.954,A -85,B 0,C 180,E1 -26881.737,E2 -26881.737} C_VEL
LIN {X 0,Y 106.021,Z 449.915,A -85,B 0,C 180,E1 -26885.684,E2 -26885.684} C_VEL
LIN {X 0,Y 110.153,Z 459.658,A -85,B 0,C 180,E1 -26891.398,E2 -26891.398} C_VEL
LIN {X 0,Y 112.128,Z 466.205,A -85,B 0,C 180,E1 -26894.892,E2 -26894.892} C_VEL
LIN {X 0,Y 112.694,Z 471.978,A -85,B 0,C 180,E1 -26897.599,E2 -26897.599} C_VEL
LIN {X 0,Y 112.842,Z 477.261,A -85,B 0,C 180,E1 -26900.139,E2 -26900.139} C_VEL
LIN {X 0,Y 112.166,Z 479.387,A -85,B 0,C 180,E1 -26900.989,E2 -26900.989} C_VEL
LIN {X 0,Y 107.19,Z 489.818,A -85,B 0,C 180,E1 -26905.3,E2 -26905.3} C_VEL
LIN {X 0,Y 102.733,Z 498.275,A -85,B 0,C 180,E1 -26910.001,E2 -26910.001} C_VEL
LIN {X 0,Y 98.826,Z 505.545,A -85,B 0,C 180,E1 -26915.363,E2 -26915.363} C_VEL
LIN {X 0,Y 95.446,Z 511.989,A -85,B 0,C 180,E1 -26921.683,E2 -26921.683} C_VEL
LIN {X 0,Y 93.334,Z 516.478,A -85,B 0,C 180,E1 -26927.53,E2 -26927.53} C_VEL
LIN {X 0,Y 91.918,Z 519.953,A -85,B 0,C 180,E1 -26933.433,E2 -26933.433} C_VEL
LIN {X 0,Y 91.095,Z 523.478,A -85,B 0,C 180,E1 -26941.933,E2 -26941.933} C_VEL
LIN {X 0,Y 91.995,Z 525.421,A -85,B 0,C 180,E1 -26950.185,E2 -26950.185} C_VEL
LIN {X 0,Y 94.418,Z 526.011,A -85,B 0,C 180,E1 -26958.103,E2 -26958.103} C_VEL
LIN {X 0,Y 97.893,Z 525.419,A -85,B 0,C 180,E1 -26964.946,E2 -26964.946} C_VEL
LIN {X 0,Y 103.315,Z 523.408,A -85,B 0,C 180,E1 -26972.168,E2 -26972.168} C_VEL
LIN {X 0,Y 109.949,Z 519.917,A -85,B 0,C 180,E1 -26978.499,E2 -26978.499} C_VEL
LIN {X 0,Y 117.188,Z 515.262,A -85,B 0,C 180,E1 -26983.647,E2 -26983.647} C_VEL
LIN {X 0,Y 124.11,Z 510,A -85,B 0,C 180,E1 -26987.638,E2 -26987.638} C_VEL
LIN {X 0,Y 132.213,Z 502.756,A -85,B 0,C 180,E1 -26991.505,E2 -26991.505} C_VEL
LIN {X 0,Y 133.379,Z 501.294,A -85,B 0,C 180,E1 -26992.43,E2 -26992.43} C_VEL
LIN {X 0,Y 134.383,Z 498.46,A -85,B 0,C 180,E1 -26995.499,E2 -26995.499} C_VEL
LIN {X 0,Y 135.176,Z 495.114,A -85,B 0,C 180,E1 -27000,E2 -27000} C_VEL
LIN {X 0,Y 135.415,Z 493.43,A -85,B 0,C 180,E1 -27002.975,E2 -27002.975} C_VEL
LIN {X 0,Y 135.607,Z 492.08,A -85,B 0,C 180,E1 -27005.949,E2 -27005.949} C_VEL
LIN {X 0,Y 135.354,Z 491.492,A -85,B 0,C 180,E1 -27009.413,E2 -27009.413} C_VEL
LIN {X 0,Y 134.772,Z 491.959,A -85,B 0,C 180,E1 -27015.113,E2 -27015.113} C_VEL
LIN {X 0,Y 134.588,Z 493.28,A -85,B 0,C 180,E1 -27019.96,E2 -27019.96} C_VEL
LIN {X 0,Y 134.214,Z 495.892,A -85,B 0,C 180,E1 -27024.766,E2 -27024.766} C_VEL
LIN {X 0,Y 133.828,Z 498.453,A -85,B 0,C 180,E1 -27028.205,E2 -27028.205} C_VEL
LIN {X 0,Y 133.044,Z 502.242,A -85,B 0,C 180,E1 -27032.308,E2 -27032.308} C_VEL
LIN {X 0,Y 132.263,Z 504.689,A -85,B 0,C 180,E1 -27034.552,E2 -27034.552} C_VEL
LIN {X 0,Y 127.945,Z 510.665,A -85,B 0,C 180,E1 -27038.103,E2 -27038.103} C_VEL
LIN {X 0,Y 123.681,Z 515.516,A -85,B 0,C 180,E1 -27041.157,E2 -27041.157} C_VEL
LIN {X 0,Y 117.966,Z 520.505,A -85,B 0,C 180,E1 -27044.363,E2 -27044.363} C_VEL
LIN {X 0,Y 111.396,Z 525.477,A -85,B 0,C 180,E1 -27048.513,E2 -27048.513} C_VEL
LIN {X 0,Y 103.999,Z 530.503,A -85,B 0,C 180,E1 -27054.941,E2 -27054.941} C_VEL
LIN {X 0,Y 99.285,Z 533.173,A -85,B 0,C 180,E1 -27060.297,E2 -27060.297} C_VEL
LIN {X 0,Y 94.553,Z 535.426,A -85,B 0,C 180,E1 -27068.182,E2 -27068.182} C_VEL
LIN {X 0,Y 92.003,Z 536.163,A -85,B 0,C 180,E1 -27076.751,E2 -27076.751} C_VEL
LIN {X 0,Y 91.364,Z 535.44,A -85,B 0,C 180,E1 -27085.587,E2 -27085.587} C_VEL
LIN {X 0,Y 91.711,Z 534.504,A -85,B 0,C 180,E1 -27089.999,E2 -27089.999} C_VEL
LIN {X 0,Y 91.479,Z 533.03,A -85,B 0,C 180,E1 -27094.405,E2 -27094.405} C_VEL
LIN {X 0,Y 91.876,Z 530.007,A -85,B 0,C 180,E1 -27101.024,E2 -27101.024} C_VEL
LIN {X 0,Y 93.206,Z 525.888,A -85,B 0,C 180,E1 -27107.553,E2 -27107.553} C_VEL
LIN {X 0,Y 96.185,Z 519.58,A -85,B 0,C 180,E1 -27114.842,E2 -27114.842} C_VEL
LIN {X 0,Y 99.799,Z 512.68,A -85,B 0,C 180,E1 -27120.699,E2 -27120.699} C_VEL
LIN {X 0,Y 104.44,Z 503.929,A -85,B 0,C 180,E1 -27126.147,E2 -27126.147} C_VEL
LIN {X 0,Y 105.957,Z 500.668,A -85,B 0,C 180,E1 -27127.844,E2 -27127.844} C_VEL
LIN {X 0,Y 107.889,Z 491.357,A -85,B 0,C 180,E1 -27132.474,E2 -27132.474} C_VEL
LIN {X 0,Y 109.462,Z 480.791,A -85,B 0,C 180,E1 -27136.911,E2 -27136.911} C_VEL
LIN {X 0,Y 110.347,Z 469.964,A -85,B 0,C 180,E1 -27140.866,E2 -27140.866} C_VEL
LIN {X 0,Y 108.984,Z 463.358,A -85,B 0,C 180,E1 -27143.762,E2 -27143.762} C_VEL
LIN {X 0,Y 106.123,Z 454.476,A -85,B 0,C 180,E1 -27148.008,E2 -27148.008} C_VEL
LIN {X 0,Y 102.134,Z 444.652,A -85,B 0,C 180,E1 -27153.253,E2 -27153.253} C_VEL
LIN {X 0,Y 99.92,Z 439.927,A -85,B 0,C 180,E1 -27156.085,E2 -27156.085} C_VEL
LIN {X 0,Y 97.883,Z 436.049,A -85,B 0,C 180,E1 -27158.71,E2 -27158.71} C_VEL
LIN {X 0,Y 97.222,Z 434.501,A -85,B 0,C 180,E1 -27159.642,E2 -27159.642} C_VEL
LIN {X 0,Y 94.482,Z 430.971,A -85,B 0,C 180,E1 -27163.145,E2 -27163.145} C_VEL
LIN {X 0,Y 93.902,Z 428.789,A -85,B 0,C 180,E1 -27164.405,E2 -27164.405} C_VEL
LIN {X 0,Y 94.063,Z 428.768,A -85,B 0,C 180,E1 -27167.048,E2 -27167.048} C_VEL
LIN {X 0,Y 94.171,Z 428.75,A -85,B 0,C 180,E1 -27171.416,E2 -27171.416} C_VEL
LIN {X 0,Y 94.788,Z 428.674,A -85,B 0,C 180,E1 -27180,E2 -27180} C_VEL
LIN {X 0,Y 94.197,Z 428.751,A -85,B 0,C 180,E1 -27188.582,E2 -27188.582} C_VEL
LIN {X 0,Y 94.04,Z 428.748,A -85,B 0,C 180,E1 -27193.71,E2 -27193.71} C_VEL
LIN {X 0,Y 93.689,Z 428.793,A -85,B 0,C 180,E1 -27202.029,E2 -27202.029} C_VEL
LIN {X 0,Y 93.621,Z 428.821,A -85,B 0,C 180,E1 -27206.771,E2 -27206.771} C_VEL
LIN {X 0,Y 93.597,Z 428.812,A -85,B 0,C 180,E1 -27214.317,E2 -27214.317} C_VEL
LIN {X 0,Y 93.538,Z 428.819,A -85,B 0,C 180,E1 -27222.55,E2 -27222.55} C_VEL
LIN {X 0,Y 93.578,Z 428.978,A -85,B 0,C 180,E1 -27229.167,E2 -27229.167} C_VEL
LIN {X 0,Y 94.625,Z 431.681,A -85,B 0,C 180,E1 -27231.129,E2 -27231.129} C_VEL
LIN {X 0,Y 96.844,Z 433.895,A -85,B 0,C 180,E1 -27233.912,E2 -27233.912} C_VEL
LIN {X 0,Y 98.858,Z 437.512,A -85,B 0,C 180,E1 -27236.741,E2 -27236.741} C_VEL
LIN {X 0,Y 99.75,Z 438.472,A -85,B 0,C 180,E1 -27237.724,E2 -27237.724} C_VEL
LIN {X 0,Y 102.856,Z 443.954,A -85,B 0,C 180,E1 -27241.737,E2 -27241.737} C_VEL
LIN {X 0,Y 104.276,Z 448.001,A -85,B 0,C 180,E1 -27243.99,E2 -27243.99} C_VEL
LIN {X 0,Y 104.985,Z 452.572,A -85,B 0,C 180,E1 -27246.038,E2 -27246.038} C_VEL
LIN {X 0,Y 105.474,Z 465.181,A -85,B 0,C 180,E1 -27251.458,E2 -27251.458} C_VEL
LIN {X 0,Y 105.912,Z 468.043,A -85,B 0,C 180,E1 -27252.97,E2 -27252.97} C_VEL
LIN {X 0,Y 106.461,Z 472.15,A -85,B 0,C 180,E1 -27255.18,E2 -27255.18} C_VEL
LIN {X 0,Y 106.509,Z 478.739,A -85,B 0,C 180,E1 -27258.584,E2 -27258.584} C_VEL
LIN {X 0,Y 102.403,Z 487.315,A -85,B 0,C 180,E1 -27262.112,E2 -27262.112} C_VEL
LIN {X 0,Y 97.539,Z 496.295,A -85,B 0,C 180,E1 -27266.903,E2 -27266.903} C_VEL
LIN {X 0,Y 93.329,Z 503.693,A -85,B 0,C 180,E1 -27272.159,E2 -27272.159} C_VEL
LIN {X 0,Y 89.309,Z 510.866,A -85,B 0,C 180,E1 -27279.056,E2 -27279.056} C_VEL
LIN {X 0,Y 86.412,Z 516.511,A -85,B 0,C 180,E1 -27286.561,E2 -27286.561} C_VEL
LIN {X 0,Y 84.588,Z 520.845,A -85,B 0,C 180,E1 -27294.547,E2 -27294.547} C_VEL
LIN {X 0,Y 84.026,Z 524.053,A -85,B 0,C 180,E1 -27303.236,E2 -27303.236} C_VEL
LIN {X 0,Y 85.256,Z 525.918,A -85,B 0,C 180,E1 -27312.105,E2 -27312.105} C_VEL
LIN {X 0,Y 88.023,Z 526.472,A -85,B 0,C 180,E1 -27320.301,E2 -27320.301} C_VEL
LIN {X 0,Y 92.084,Z 525.852,A -85,B 0,C 180,E1 -27327.706,E2 -27327.706} C_VEL
LIN {X 0,Y 97.326,Z 524.116,A -85,B 0,C 180,E1 -27334.324,E2 -27334.324} C_VEL
LIN {X 0,Y 104.254,Z 520.933,A -85,B 0,C 180,E1 -27340.695,E2 -27340.695} C_VEL
LIN {X 0,Y 112.725,Z 515.955,A -85,B 0,C 180,E1 -27346.417,E2 -27346.417} C_VEL
LIN {X 0,Y 121.015,Z 510.022,A -85,B 0,C 180,E1 -27350.852,E2 -27350.852} C_VEL
LIN {X 0,Y 127.347,Z 504.691,A -85,B 0,C 180,E1 -27353.663,E2 -27353.663} C_VEL
LIN {X 0,Y 128.399,Z 503.102,A -85,B 0,C 180,E1 -27355.272,E2 -27355.272} C_VEL
LIN {X 0,Y 129.614,Z 499.827,A -85,B 0,C 180,E1 -27360,E2 -27360} C_VEL
LIN {X 0,Y 130.069,Z 498.218,A -85,B 0,C 180,E1 -27363.097,E2 -27363.097} C_VEL
LIN {X 0,Y 130.424,Z 496.927,A -85,B 0,C 180,E1 -27366.187,E2 -27366.187} C_VEL
LIN {X 0,Y 130.275,Z 496.452,A -85,B 0,C 180,E1 -27369.314,E2 -27369.314} C_VEL
LIN {X 0,Y 129.842,Z 496.664,A -85,B 0,C 180,E1 -27373.021,E2 -27373.021} C_VEL
LIN {X 0,Y 129.476,Z 497.93,A -85,B 0,C 180,E1 -27379.007,E2 -27379.007} C_VEL
LIN {X 0,Y 128.939,Z 500.396,A -85,B 0,C 180,E1 -27384.129,E2 -27384.129} C_VEL
LIN {X 0,Y 128.487,Z 502.232,A -85,B 0,C 180,E1 -27386.941,E2 -27386.941} C_VEL
LIN {X 0,Y 127.364,Z 505.957,A -85,B 0,C 180,E1 -27391.389,E2 -27391.389} C_VEL
LIN {X 0,Y 126.898,Z 507.127,A -85,B 0,C 180,E1 -27392.631,E2 -27392.631} C_VEL
LIN {X 0,Y 124.455,Z 510.265,A -85,B 0,C 180,E1 -27394.742,E2 -27394.742} C_VEL
LIN {X 0,Y 120.14,Z 514.973,A -85,B 0,C 180,E1 -27397.84,E2 -27397.84} C_VEL
LIN {X 0,Y 117.959,Z 517.045,A -85,B 0,C 180,E1 -27399.237,E2 -27399.237} C_VEL
LIN {X 0,Y 110.73,Z 522.565,A -85,B 0,C 180,E1 -27403.122,E2 -27403.122} C_VEL
LIN {X 0,Y 104.042,Z 527.003,A -85,B 0,C 180,E1 -27407.507,E2 -27407.507} C_VEL
LIN {X 0,Y 96.458,Z 531.403,A -85,B 0,C 180,E1 -27414.346,E2 -27414.346} C_VEL
LIN {X 0,Y 90.321,Z 534.248,A -85,B 0,C 180,E1 -27422.168,E2 -27422.168} C_VEL
LIN {X 0,Y 86.252,Z 535.567,A -85,B 0,C 180,E1 -27430.977,E2 -27430.977} C_VEL
LIN {X 0,Y 84.414,Z 535.458,A -85,B 0,C 180,E1 -27440.414,E2 -27440.414} C_VEL
LIN {X 0,Y 84.415,Z 534.382,A -85,B 0,C 180,E1 -27447.51,E2 -27447.51} C_VEL
LIN {X 0,Y 84.646,Z 533.804,A -85,B 0,C 180,E1 -27449.999,E2 -27449.999} C_VEL
LIN {X 0,Y 84.414,Z 532.265,A -85,B 0,C 180,E1 -27454.774,E2 -27454.774} C_VEL
LIN {X 0,Y 84.907,Z 529.111,A -85,B 0,C 180,E1 -27461.941,E2 -27461.941} C_VEL
LIN {X 0,Y 86.447,Z 524.855,A -85,B 0,C 180,E1 -27468.976,E2 -27468.976} C_VEL
LIN {X 0,Y 89.186,Z 519.401,A -85,B 0,C 180,E1 -27475.682,E2 -27475.682} C_VEL
LIN {X 0,Y 92.996,Z 512.565,A -85,B 0,C 180,E1 -27481.937,E2 -27481.937} C_VEL
LIN {X 0,Y 97.367,Z 504.829,A -85,B 0,C 180,E1 -27487.186,E2 -27487.186} C_VEL
LIN {X 0,Y 99.462,Z 500.686,A -85,B 0,C 180,E1 -27489.488,E2 -27489.488} C_VEL
LIN {X 0,Y 101.381,Z 492.531,A -85,B 0,C 180,E1 -27493.884,E2 -27493.884} C_VEL
LIN {X 0,Y 103.224,Z 482.413,A -85,B 0,C 180,E1 -27498.496,E2 -27498.496} C_VEL
LIN {X 0,Y 104.368,Z 471.916,A -85,B 0,C 180,E1 -27502.696,E2 -27502.696} C_VEL
LIN {X 0,Y 103.206,Z 466.089,A -85,B 0,C 180,E1 -27505.554,E2 -27505.554} C_VEL
LIN {X 0,Y 100.387,Z 456.565,A -85,B 0,C 180,E1 -27510.656,E2 -27510.656} C_VEL
LIN {X 0,Y 97.461,Z 448.912,A -85,B 0,C 180,E1 -27515.28,E2 -27515.28} C_VEL
LIN {X 0,Y 95.686,Z 444.784,A -85,B 0,C 180,E1 -27518.03,E2 -27518.03} C_VEL
LIN {X 0,Y 93.559,Z 439.956,A -85,B 0,C 180,E1 -27521.524,E2 -27521.524} C_VEL
LIN {X 0,Y 91.206,Z 436.353,A -85,B 0,C 180,E1 -27525.141,E2 -27525.141} C_VEL
LIN {X 0,Y 90.668,Z 435.046,A -85,B 0,C 180,E1 -27526.197,E2 -27526.197} C_VEL
LIN {X 0,Y 88.227,Z 432.769,A -85,B 0,C 180,E1 -27530.11,E2 -27530.11} C_VEL
LIN {X 0,Y 87.111,Z 429.617,A -85,B 0,C 180,E1 -27533.05,E2 -27533.05} C_VEL
LIN {X 0,Y 87.714,Z 429.554,A -85,B 0,C 180,E1 -27540,E2 -27540} C_VEL
LIN {X 0,Y 87.105,Z 429.631,A -85,B 0,C 180,E1 -27549.287,E2 -27549.287} C_VEL
LIN {X 0,Y 86.948,Z 429.632,A -85,B 0,C 180,E1 -27554.088,E2 -27554.088} C_VEL
LIN {X 0,Y 86.659,Z 429.689,A -85,B 0,C 180,E1 -27558.93,E2 -27558.93} C_VEL
LIN {X 0,Y 86.583,Z 429.697,A -85,B 0,C 180,E1 -27566.768,E2 -27566.768} C_VEL
LIN {X 0,Y 86.515,Z 429.703,A -85,B 0,C 180,E1 -27575.678,E2 -27575.678} C_VEL
LIN {X 0,Y 86.445,Z 429.769,A -85,B 0,C 180,E1 -27579.722,E2 -27579.722} C_VEL
LIN {X 0,Y 87.421,Z 432.43,A -85,B 0,C 180,E1 -27582.537,E2 -27582.537} C_VEL
LIN {X 0,Y 89.418,Z 434.641,A -85,B 0,C 180,E1 -27586.229,E2 -27586.229} C_VEL
LIN {X 0,Y 90.537,Z 435.546,A -85,B 0,C 180,E1 -27587.941,E2 -27587.941} C_VEL
LIN {X 0,Y 92.057,Z 438.604,A -85,B 0,C 180,E1 -27590.872,E2 -27590.872} C_VEL
LIN {X 0,Y 93.579,Z 440.351,A -85,B 0,C 180,E1 -27593.074,E2 -27593.074} C_VEL
LIN {X 0,Y 94.57,Z 442.444,A -85,B 0,C 180,E1 -27594.833,E2 -27594.833} C_VEL
LIN {X 0,Y 96.409,Z 445.242,A -85,B 0,C 180,E1 -27597.445,E2 -27597.445} C_VEL
LIN {X 0,Y 99.779,Z 451.717,A -85,B 0,C 180,E1 -27602.512,E2 -27602.512} C_VEL
LIN {X 0,Y 102.505,Z 458.118,A -85,B 0,C 180,E1 -27606.824,E2 -27606.824} C_VEL
LIN {X 0,Y 105.13,Z 465.119,A -85,B 0,C 180,E1 -27611.259,E2 -27611.259} C_VEL
LIN {X 0,Y 105.912,Z 468.043,A -85,B 0,C 180,E1 -27612.97,E2 -27612.97} C_VEL
LIN {X 0,Y 105.799,Z 470.996,A -85,B 0,C 180,E1 -27614.312,E2 -27614.312} C_VEL
LIN {X 0,Y 104.567,Z 474.198,A -85,B 0,C 180,E1 -27615.382,E2 -27615.382} C_VEL
LIN {X 0,Y 98.399,Z 483.849,A -85,B 0,C 180,E1 -27618.302,E2 -27618.302} C_VEL
LIN {X 0,Y 97.828,Z 484.879,A -85,B 0,C 180,E1 -27618.737,E2 -27618.737} C_VEL
LIN {X 0,Y 92.91,Z 493.712,A -85,B 0,C 180,E1 -27623.183,E2 -27623.183} C_VEL
LIN {X 0,Y 87.913,Z 502.048,A -85,B 0,C 180,E1 -27628.856,E2 -27628.856} C_VEL
LIN {X 0,Y 83.336,Z 509.632,A -85,B 0,C 180,E1 -27636.052,E2 -27636.052} C_VEL
LIN {X 0,Y 79.827,Z 515.938,A -85,B 0,C 180,E1 -27644.427,E2 -27644.427} C_VEL
LIN {X 0,Y 78.041,Z 519.615,A -85,B 0,C 180,E1 -27651.115,E2 -27651.115} C_VEL
LIN {X 0,Y 76.932,Z 523.255,A -85,B 0,C 180,E1 -27660.162,E2 -27660.162} C_VEL
LIN {X 0,Y 77.546,Z 525.626,A -85,B 0,C 180,E1 -27669.377,E2 -27669.377} C_VEL
LIN {X 0,Y 78.937,Z 526.537,A -85,B 0,C 180,E1 -27675.42,E2 -27675.42} C_VEL
LIN {X 0,Y 81.875,Z 526.933,A -85,B 0,C 180,E1 -27683.067,E2 -27683.067} C_VEL
LIN {X 0,Y 87.481,Z 526.082,A -85,B 0,C 180,E1 -27692.094,E2 -27692.094} C_VEL
LIN {X 0,Y 92.404,Z 524.535,A -85,B 0,C 180,E1 -27697.648,E2 -27697.648} C_VEL
LIN {X 0,Y 99.3,Z 521.652,A -85,B 0,C 180,E1 -27703.554,E2 -27703.554} C_VEL
LIN {X 0,Y 107.461,Z 517.308,A -85,B 0,C 180,E1 -27708.815,E2 -27708.815} C_VEL
LIN {X 0,Y 115.667,Z 511.975,A -85,B 0,C 180,E1 -27713.02,E2 -27713.02} C_VEL
LIN {X 0,Y 122.243,Z 506.996,A -85,B 0,C 180,E1 -27715.853,E2 -27715.853} C_VEL
LIN {X 0,Y 122.762,Z 506.27,A -85,B 0,C 180,E1 -27716.718,E2 -27716.718} C_VEL
LIN {X 0,Y 123.786,Z 504.274,A -85,B 0,C 180,E1 -27720,E2 -27720} C_VEL
LIN {X 0,Y 124.452,Z 502.714,A -85,B 0,C 180,E1 -27723.237,E2 -27723.237} C_VEL
LIN {X 0,Y 125.006,Z 501.503,A -85,B 0,C 180,E1 -27726.456,E2 -27726.456} C_VEL
LIN {X 0,Y 124.861,Z 501.162,A -85,B 0,C 180,E1 -27729.721,E2 -27729.721} C_VEL
LIN {X 0,Y 124.497,Z 501.384,A -85,B 0,C 180,E1 -27733.05,E2 -27733.05} C_VEL
LIN {X 0,Y 124.216,Z 501.972,A -85,B 0,C 180,E1 -27736.433,E2 -27736.433} C_VEL
LIN {X 0,Y 123.87,Z 503.033,A -85,B 0,C 180,E1 -27739.902,E2 -27739.902} C_VEL
LIN {X 0,Y 123.289,Z 505.057,A -85,B 0,C 180,E1 -27744.208,E2 -27744.208} C_VEL
LIN {X 0,Y 122.15,Z 508.032,A -85,B 0,C 180,E1 -27748.671,E2 -27748.671} C_VEL
LIN {X 0,Y 121.694,Z 509.089,A -85,B 0,C 180,E1 -27749.972,E2 -27749.972} C_VEL
LIN {X 0,Y 120.752,Z 510.618,A -85,B 0,C 180,E1 -27751.588,E2 -27751.588} C_VEL
LIN {X 0,Y 115.813,Z 515.54,A -85,B 0,C 180,E1 -27754.992,E2 -27754.992} C_VEL
LIN {X 0,Y 113.552,Z 517.492,A -85,B 0,C 180,E1 -27756.428,E2 -27756.428} C_VEL
LIN {X 0,Y 106.016,Z 522.824,A -85,B 0,C 180,E1 -27760.328,E2 -27760.328} C_VEL
LIN {X 0,Y 98.919,Z 527.102,A -85,B 0,C 180,E1 -27764.726,E2 -27764.726} C_VEL
LIN {X 0,Y 90.774,Z 531.339,A -85,B 0,C 180,E1 -27771.728,E2 -27771.728} C_VEL
LIN {X 0,Y 84.081,Z 533.969,A -85,B 0,C 180,E1 -27779.899,E2 -27779.899} C_VEL
LIN {X 0,Y 79.546,Z 535.161,A -85,B 0,C 180,E1 -27789.303,E2 -27789.303} C_VEL
LIN {X 0,Y 77.412,Z 534.894,A -85,B 0,C 180,E1 -27799.537,E2 -27799.537} C_VEL
LIN {X 0,Y 77.564,Z 533.094,A -85,B 0,C 180,E1 -27809.999,E2 -27809.999} C_VEL
LIN {X 0,Y 77.418,Z 530.508,A -85,B 0,C 180,E1 -27817.825,E2 -27817.825} C_VEL
LIN {X 0,Y 78.404,Z 526.869,A -85,B 0,C 180,E1 -27825.598,E2 -27825.598} C_VEL
LIN {X 0,Y 80.589,Z 522.076,A -85,B 0,C 180,E1 -27833.104,E2 -27833.104} C_VEL
LIN {X 0,Y 84.13,Z 516.029,A -85,B 0,C 180,E1 -27840.079,E2 -27840.079} C_VEL
LIN {X 0,Y 88.659,Z 508.47,A -85,B 0,C 180,E1 -27846.477,E2 -27846.477} C_VEL
LIN {X 0,Y 92.708,Z 501.496,A -85,B 0,C 180,E1 -27850.879,E2 -27850.879} C_VEL
LIN {X 0,Y 94.926,Z 493.673,A -85,B 0,C 180,E1 -27855.444,E2 -27855.444} C_VEL
LIN {X 0,Y 97.04,Z 483.95,A -85,B 0,C 180,E1 -27860.282,E2 -27860.282} C_VEL
LIN {X 0,Y 98.421,Z 474.411,A -85,B 0,C 180,E1 -27864.435,E2 -27864.435} C_VEL
LIN {X 0,Y 97.103,Z 467.382,A -85,B 0,C 180,E1 -27868.35,E2 -27868.35} C_VEL
LIN {X 0,Y 95.321,Z 460.524,A -85,B 0,C 180,E1 -27872.443,E2 -27872.443} C_VEL
LIN {X 0,Y 92.169,Z 451.097,A -85,B 0,C 180,E1 -27878.765,E2 -27878.765} C_VEL
LIN {X 0,Y 90.221,Z 446.006,A -85,B 0,C 180,E1 -27882.724,E2 -27882.724} C_VEL
LIN {X 0,Y 87.849,Z 441.782,A -85,B 0,C 180,E1 -27887.11,E2 -27887.11} C_VEL
LIN {X 0,Y 87.375,Z 441.031,A -85,B 0,C 180,E1 -27888.055,E2 -27888.055} C_VEL
LIN {X 0,Y 85.38,Z 438.599,A -85,B 0,C 180,E1 -27892.048,E2 -27892.048} C_VEL
LIN {X 0,Y 84.452,Z 436.165,A -85,B 0,C 180,E1 -27894.794,E2 -27894.794} C_VEL
LIN {X 0,Y 81.896,Z 433.986,A -85,B 0,C 180,E1 -27901.845,E2 -27901.845} C_VEL
LIN {X 0,Y 80.138,Z 431.585,A -85,B 0,C 180,E1 -27911.856,E2 -27911.856} C_VEL
LIN {X 0,Y 79.944,Z 431.421,A -85,B 0,C 180,E1 -27915.292,E2 -27915.292} C_VEL
LIN {X 0,Y 80.208,Z 432.815,A -85,B 0,C 180,E1 -27924.596,E2 -27924.596} C_VEL
LIN {X 0,Y 83.91,Z 436.565,A -85,B 0,C 180,E1 -27938.547,E2 -27938.547} C_VEL
LIN {X 0,Y 85.484,Z 439.975,A -85,B 0,C 180,E1 -27943.232,E2 -27943.232} C_VEL
LIN {X 0,Y 87.218,Z 441.545,A -85,B 0,C 180,E1 -27946.488,E2 -27946.488} C_VEL
LIN {X 0,Y 88.928,Z 444.9,A -85,B 0,C 180,E1 -27950.182,E2 -27950.182} C_VEL
LIN {X 0,Y 89.738,Z 445.903,A -85,B 0,C 180,E1 -27951.552,E2 -27951.552} C_VEL
LIN {X 0,Y 92.484,Z 451.178,A -85,B 0,C 180,E1 -27956.711,E2 -27956.711} C_VEL
LIN {X 0,Y 95.456,Z 457.561,A -85,B 0,C 180,E1 -27962.07,E2 -27962.07} C_VEL
LIN {X 0,Y 97.851,Z 464.086,A -85,B 0,C 180,E1 -27966.819,E2 -27966.819} C_VEL
LIN {X 0,Y 99.788,Z 470.208,A -85,B 0,C 180,E1 -27971.017,E2 -27971.017} C_VEL
LIN {X 0,Y 100.389,Z 474.711,A -85,B 0,C 180,E1 -27973.739,E2 -27973.739} C_VEL
LIN {X 0,Y 100.234,Z 480.19,A -85,B 0,C 180,E1 -27976.829,E2 -27976.829} C_VEL
LIN {X 0,Y 97.828,Z 484.879,A -85,B 0,C 180,E1 -27978.737,E2 -27978.737} C_VEL
LIN {X 0,Y 96.065,Z 487.753,A -85,B 0,C 180,E1 -27979.943,E2 -27979.943} C_VEL
LIN {X 0,Y 91.399,Z 493.122,A -85,B 0,C 180,E1 -27982.075,E2 -27982.075} C_VEL
LIN {X 0,Y 82.507,Z 501.568,A -85,B 0,C 180,E1 -27986.439,E2 -27986.439} C_VEL
LIN {X 0,Y 79.736,Z 504.974,A -85,B 0,C 180,E1 -27989.24,E2 -27989.24} C_VEL
LIN {X 0,Y 75.488,Z 511.646,A -85,B 0,C 180,E1 -27996.684,E2 -27996.684} C_VEL
LIN {X 0,Y 72.552,Z 516.68,A -85,B 0,C 180,E1 -28004.374,E2 -28004.374} C_VEL
LIN {X 0,Y 70.467,Z 521.037,A -85,B 0,C 180,E1 -28013.513,E2 -28013.513} C_VEL
LIN {X 0,Y 69.829,Z 523.41,A -85,B 0,C 180,E1 -28020.215,E2 -28020.215} C_VEL
LIN {X 0,Y 70.101,Z 525.208,A -85,B 0,C 180,E1 -28026.981,E2 -28026.981} C_VEL
LIN {X 0,Y 72.146,Z 526.901,A -85,B 0,C 180,E1 -28037.007,E2 -28037.007} C_VEL
LIN {X 0,Y 75.994,Z 527.395,A -85,B 0,C 180,E1 -28046.339,E2 -28046.339} C_VEL
LIN {X 0,Y 81.264,Z 526.737,A -85,B 0,C 180,E1 -28054.378,E2 -28054.378} C_VEL
LIN {X 0,Y 88.64,Z 524.691,A -85,B 0,C 180,E1 -28062.073,E2 -28062.073} C_VEL
LIN {X 0,Y 97.375,Z 521.128,A -85,B 0,C 180,E1 -28068.53,E2 -28068.53} C_VEL
LIN {X 0,Y 106.126,Z 516.565,A -85,B 0,C 180,E1 -28073.386,E2 -28073.386} C_VEL
LIN {X 0,Y 114.355,Z 511.333,A -85,B 0,C 180,E1 -28077.025,E2 -28077.025} C_VEL
LIN {X 0,Y 117.034,Z 509.338,A -85,B 0,C 180,E1 -28078.279,E2 -28078.279} C_VEL
LIN {X 0,Y 117.651,Z 508.436,A -85,B 0,C 180,E1 -28080,E2 -28080} C_VEL
LIN {X 0,Y 118.611,Z 506.92,A -85,B 0,C 180,E1 -28083.397,E2 -28083.397} C_VEL
LIN {X 0,Y 119.359,Z 505.786,A -85,B 0,C 180,E1 -28086.763,E2 -28086.763} C_VEL
LIN {X 0,Y 119.198,Z 505.603,A -85,B 0,C 180,E1 -28090.188,E2 -28090.188} C_VEL
LIN {X 0,Y 118.833,Z 505.901,A -85,B 0,C 180,E1 -28093.684,E2 -28093.684} C_VEL
LIN {X 0,Y 118.36,Z 506.901,A -85,B 0,C 180,E1 -28098.187,E2 -28098.187} C_VEL
LIN {X 0,Y 117.953,Z 507.855,A -85,B 0,C 180,E1 -28100.946,E2 -28100.946} C_VEL
LIN {X 0,Y 116.914,Z 510.184,A -85,B 0,C 180,E1 -28105.62,E2 -28105.62} C_VEL
LIN {X 0,Y 115.611,Z 512.534,A -85,B 0,C 180,E1 -28109.099,E2 -28109.099} C_VEL
LIN {X 0,Y 112.969,Z 515.1,A -85,B 0,C 180,E1 -28111.195,E2 -28111.195} C_VEL
LIN {X 0,Y 109.405,Z 518.003,A -85,B 0,C 180,E1 -28113.374,E2 -28113.374} C_VEL
LIN {X 0,Y 104.213,Z 521.51,A -85,B 0,C 180,E1 -28115.976,E2 -28115.976} C_VEL
LIN {X 0,Y 96.469,Z 525.955,A -85,B 0,C 180,E1 -28120.097,E2 -28120.097} C_VEL
LIN {X 0,Y 89.48,Z 529.432,A -85,B 0,C 180,E1 -28125.018,E2 -28125.018} C_VEL
LIN {X 0,Y 81.386,Z 532.646,A -85,B 0,C 180,E1 -28132.808,E2 -28132.808} C_VEL
LIN {X 0,Y 75.099,Z 534.403,A -85,B 0,C 180,E1 -28142.1,E2 -28142.1} C_VEL
LIN {X 0,Y 71.363,Z 534.706,A -85,B 0,C 180,E1 -28152.815,E2 -28152.815} C_VEL
LIN {X 0,Y 70.163,Z 533.521,A -85,B 0,C 180,E1 -28164.25,E2 -28164.25} C_VEL
LIN {X 0,Y 70.476,Z 532.368,A -85,B 0,C 180,E1 -28169.999,E2 -28169.999} C_VEL
LIN {X 0,Y 70.392,Z 529.644,A -85,B 0,C 180,E1 -28178.612,E2 -28178.612} C_VEL
LIN {X 0,Y 71.579,Z 525.859,A -85,B 0,C 180,E1 -28187.129,E2 -28187.129} C_VEL
LIN {X 0,Y 74.095,Z 520.919,A -85,B 0,C 180,E1 -28195.265,E2 -28195.265} C_VEL
LIN {X 0,Y 78.051,Z 514.712,A -85,B 0,C 180,E1 -28202.699,E2 -28202.699} C_VEL
LIN {X 0,Y 83.029,Z 506.89,A -85,B 0,C 180,E1 -28209.405,E2 -28209.405} C_VEL
LIN {X 0,Y 86.36,Z 501.526,A -85,B 0,C 180,E1 -28212.911,E2 -28212.911} C_VEL
LIN {X 0,Y 88.531,Z 494.658,A -85,B 0,C 180,E1 -28217.246,E2 -28217.246} C_VEL
LIN {X 0,Y 90.947,Z 485.178,A -85,B 0,C 180,E1 -28222.373,E2 -28222.373} C_VEL
LIN {X 0,Y 92.449,Z 477.564,A -85,B 0,C 180,E1 -28226.002,E2 -28226.002} C_VEL
LIN {X 0,Y 91.885,Z 472.277,A -85,B 0,C 180,E1 -28229.176,E2 -28229.176} C_VEL
LIN {X 0,Y 90.093,Z 464.053,A -85,B 0,C 180,E1 -28234.593,E2 -28234.593} C_VEL
LIN {X 0,Y 88.029,Z 456.495,A -85,B 0,C 180,E1 -28240.166,E2 -28240.166} C_VEL
LIN {X 0,Y 86.257,Z 451.233,A -85,B 0,C 180,E1 -28244.645,E2 -28244.645} C_VEL
LIN {X 0,Y 84.504,Z 447.718,A -85,B 0,C 180,E1 -28248.648,E2 -28248.648} C_VEL
LIN {X 0,Y 82.169,Z 443.799,A -85,B 0,C 180,E1 -28254.649,E2 -28254.649} C_VEL
LIN {X 0,Y 81.713,Z 442.564,A -85,B 0,C 180,E1 -28256.302,E2 -28256.302} C_VEL
LIN {X 0,Y 79.613,Z 440.555,A -85,B 0,C 180,E1 -28263.163,E2 -28263.163} C_VEL
LIN {X 0,Y 78.336,Z 438.424,A -85,B 0,C 180,E1 -28272.21,E2 -28272.21} C_VEL
LIN {X 0,Y 78.072,Z 438.474,A -85,B 0,C 180,E1 -28277.012,E2 -28277.012} C_VEL
LIN {X 0,Y 78.415,Z 440.052,A -85,B 0,C 180,E1 -28286.045,E2 -28286.045} C_VEL
LIN {X 0,Y 81.131,Z 442.934,A -85,B 0,C 180,E1 -28297.329,E2 -28297.329} C_VEL
LIN {X 0,Y 82.166,Z 445.756,A -85,B 0,C 180,E1 -28301.363,E2 -28301.363} C_VEL
LIN {X 0,Y 83.719,Z 447.492,A -85,B 0,C 180,E1 -28305.025,E2 -28305.025} C_VEL
LIN {X 0,Y 87.312,Z 454.566,A -85,B 0,C 180,E1 -28313.605,E2 -28313.605} C_VEL
LIN {X 0,Y 89.868,Z 460.579,A -85,B 0,C 180,E1 -28319.345,E2 -28319.345} C_VEL
LIN {X 0,Y 91.902,Z 466.463,A -85,B 0,C 180,E1 -28324.24,E2 -28324.24} C_VEL
LIN {X 0,Y 93.965,Z 473.683,A -85,B 0,C 180,E1 -28329.791,E2 -28329.791} C_VEL
LIN {X 0,Y 94.276,Z 478.059,A -85,B 0,C 180,E1 -28332.653,E2 -28332.653} C_VEL
LIN {X 0,Y 93.894,Z 481.679,A -85,B 0,C 180,E1 -28334.814,E2 -28334.814} C_VEL
LIN {X 0,Y 89.229,Z 489.976,A -85,B 0,C 180,E1 -28338.645,E2 -28338.645} C_VEL
LIN {X 0,Y 84.065,Z 498.299,A -85,B 0,C 180,E1 -28343.724,E2 -28343.724} C_VEL
LIN {X 0,Y 79.736,Z 504.974,A -85,B 0,C 180,E1 -28349.24,E2 -28349.24} C_VEL
LIN {X 0,Y 77.126,Z 508.185,A -85,B 0,C 180,E1 -28352.316,E2 -28352.316} C_VEL
LIN {X 0,Y 71.478,Z 512.906,A -85,B 0,C 180,E1 -28357.442,E2 -28357.442} C_VEL
LIN {X 0,Y 66.178,Z 517.002,A -85,B 0,C 180,E1 -28363.613,E2 -28363.613} C_VEL
LIN {X 0,Y 64.282,Z 519.21,A -85,B 0,C 180,E1 -28368.171,E2 -28368.171} C_VEL
LIN {X 0,Y 62.941,Z 522.465,A -85,B 0,C 180,E1 -28376.71,E2 -28376.71} C_VEL
LIN {X 0,Y 63.187,Z 525.65,A -85,B 0,C 180,E1 -28388.868,E2 -28388.868} C_VEL
LIN {X 0,Y 65.807,Z 527.383,A -85,B 0,C 180,E1 -28400.149,E2 -28400.149} C_VEL
LIN {X 0,Y 70.327,Z 527.859,A -85,B 0,C 180,E1 -28410.021,E2 -28410.021} C_VEL
LIN {X 0,Y 76.351,Z 527.188,A -85,B 0,C 180,E1 -28418.395,E2 -28418.395} C_VEL
LIN {X 0,Y 83.592,Z 525.416,A -85,B 0,C 180,E1 -28425.39,E2 -28425.39} C_VEL
LIN {X 0,Y 92.38,Z 522.273,A -85,B 0,C 180,E1 -28431.496,E2 -28431.496} C_VEL
LIN {X 0,Y 102.912,Z 517.202,A -85,B 0,C 180,E1 -28436.915,E2 -28436.915} C_VEL
LIN {X 0,Y 110.541,Z 512.694,A -85,B 0,C 180,E1 -28440,E2 -28440} C_VEL
LIN {X 0,Y 112.75,Z 510.601,A -85,B 0,C 180,E1 -28444.197,E2 -28444.197} C_VEL
LIN {X 0,Y 113.447,Z 509.747,A -85,B 0,C 180,E1 -28447.61,E2 -28447.61} C_VEL
LIN {X 0,Y 113.294,Z 509.736,A -85,B 0,C 180,E1 -28450.725,E2 -28450.725} C_VEL
LIN {X 0,Y 112.885,Z 510.153,A -85,B 0,C 180,E1 -28454.42,E2 -28454.42} C_VEL
LIN {X 0,Y 112.427,Z 510.989,A -85,B 0,C 180,E1 -28458.213,E2 -28458.213} C_VEL
LIN {X 0,Y 111.555,Z 512.453,A -85,B 0,C 180,E1 -28462.21,E2 -28462.21} C_VEL
LIN {X 0,Y 111.096,Z 513.378,A -85,B 0,C 180,E1 -28464.28,E2 -28464.28} C_VEL
LIN {X 0,Y 110.16,Z 514.79,A -85,B 0,C 180,E1 -28466.726,E2 -28466.726} C_VEL
LIN {X 0,Y 108.106,Z 516.608,A -85,B 0,C 180,E1 -28468.641,E2 -28468.641} C_VEL
LIN {X 0,Y 102.971,Z 520.201,A -85,B 0,C 180,E1 -28471.444,E2 -28471.444} C_VEL
LIN {X 0,Y 94.705,Z 524.803,A -85,B 0,C 180,E1 -28475.284,E2 -28475.284} C_VEL
LIN {X 0,Y 86.988,Z 528.409,A -85,B 0,C 180,E1 -28479.867,E2 -28479.867} C_VEL
LIN {X 0,Y 80.058,Z 531.115,A -85,B 0,C 180,E1 -28485.389,E2 -28485.389} C_VEL
LIN {X 0,Y 72.11,Z 533.441,A -85,B 0,C 180,E1 -28494.212,E2 -28494.212} C_VEL
LIN {X 0,Y 68.879,Z 534.043,A -85,B 0,C 180,E1 -28499.324,E2 -28499.324} C_VEL
LIN {X 0,Y 64.6,Z 534.162,A -85,B 0,C 180,E1 -28510.95,E2 -28510.95} C_VEL
LIN {X 0,Y 63.114,Z 532.855,A -85,B 0,C 180,E1 -28523.605,E2 -28523.605} C_VEL
LIN {X 0,Y 63.409,Z 531.63,A -85,B 0,C 180,E1 -28529.998,E2 -28529.998} C_VEL
LIN {X 0,Y 63.372,Z 528.776,A -85,B 0,C 180,E1 -28539.574,E2 -28539.574} C_VEL
LIN {X 0,Y 64.822,Z 524.849,A -85,B 0,C 180,E1 -28548.979,E2 -28548.979} C_VEL
LIN {X 0,Y 68.363,Z 518.74,A -85,B 0,C 180,E1 -28559.228,E2 -28559.228} C_VEL
LIN {X 0,Y 72.966,Z 512.072,A -85,B 0,C 180,E1 -28567.01,E2 -28567.01} C_VEL
LIN {X 0,Y 78.689,Z 503.782,A -85,B 0,C 180,E1 -28573.8,E2 -28573.8} C_VEL
LIN {X 0,Y 80.609,Z 500.268,A -85,B 0,C 180,E1 -28576.189,E2 -28576.189} C_VEL
LIN {X 0,Y 83.563,Z 491.343,A -85,B 0,C 180,E1 -28581.987,E2 -28581.987} C_VEL
LIN {X 0,Y 85.919,Z 482.855,A -85,B 0,C 180,E1 -28586.627,E2 -28586.627} C_VEL
LIN {X 0,Y 86.625,Z 479.234,A -85,B 0,C 180,E1 -28588.488,E2 -28588.488} C_VEL
LIN {X 0,Y 85.791,Z 472.504,A -85,B 0,C 180,E1 -28593.223,E2 -28593.223} C_VEL
LIN {X 0,Y 84.301,Z 464.618,A -85,B 0,C 180,E1 -28599.249,E2 -28599.249} C_VEL
LIN {X 0,Y 83.291,Z 460.395,A -85,B 0,C 180,E1 -28602.823,E2 -28602.823} C_VEL
LIN {X 0,Y 82.285,Z 456.555,A -85,B 0,C 180,E1 -28606.416,E2 -28606.416} C_VEL
LIN {X 0,Y 81.046,Z 453.649,A -85,B 0,C 180,E1 -28610.013,E2 -28610.013} C_VEL
LIN {X 0,Y 79.388,Z 450.775,A -85,B 0,C 180,E1 -28614.922,E2 -28614.922} C_VEL
LIN {X 0,Y 78.849,Z 448.979,A -85,B 0,C 180,E1 -28617.446,E2 -28617.446} C_VEL
LIN {X 0,Y 76.708,Z 446.607,A -85,B 0,C 180,E1 -28626.203,E2 -28626.203} C_VEL
LIN {X 0,Y 76.25,Z 445.475,A -85,B 0,C 180,E1 -28630.623,E2 -28630.623} C_VEL
LIN {X 0,Y 75.929,Z 445.149,A -85,B 0,C 180,E1 -28636.122,E2 -28636.122} C_VEL
LIN {X 0,Y 75.801,Z 445.98,A -85,B 0,C 180,E1 -28642.009,E2 -28642.009} C_VEL
LIN {X 0,Y 77.984,Z 449.197,A -85,B 0,C 180,E1 -28655.802,E2 -28655.802} C_VEL
LIN {X 0,Y 79.033,Z 452.011,A -85,B 0,C 180,E1 -28660.57,E2 -28660.57} C_VEL
LIN {X 0,Y 80.316,Z 453.907,A -85,B 0,C 180,E1 -28664.431,E2 -28664.431} C_VEL
LIN {X 0,Y 82.916,Z 459.68,A -85,B 0,C 180,E1 -28672.089,E2 -28672.089} C_VEL
LIN {X 0,Y 85.108,Z 465.699,A -85,B 0,C 180,E1 -28678.413,E2 -28678.413} C_VEL
LIN {X 0,Y 86.624,Z 470.925,A -85,B 0,C 180,E1 -28683.186,E2 -28683.186} C_VEL
LIN {X 0,Y 88.107,Z 477.051,A -85,B 0,C 180,E1 -28688.435,E2 -28688.435} C_VEL
LIN {X 0,Y 88.139,Z 481.182,A -85,B 0,C 180,E1 -28691.402,E2 -28691.402} C_VEL
LIN {X 0,Y 87.659,Z 483.087,A -85,B 0,C 180,E1 -28692.505,E2 -28692.505} C_VEL
LIN {X 0,Y 82.773,Z 491.225,A -85,B 0,C 180,E1 -28696.499,E2 -28696.499} C_VEL
LIN {X 0,Y 76.8,Z 500.142,A -85,B 0,C 180,E1 -28702.47,E2 -28702.47} C_VEL
LIN {X 0,Y 71.378,Z 507.983,A -85,B 0,C 180,E1 -28710.001,E2 -28710.001} C_VEL
LIN {X 0,Y 67.001,Z 514.552,A -85,B 0,C 180,E1 -28719.054,E2 -28719.054} C_VEL
LIN {X 0,Y 64.282,Z 519.21,A -85,B 0,C 180,E1 -28728.171,E2 -28728.171} C_VEL
LIN {X 0,Y 62.709,Z 521.198,A -85,B 0,C 180,E1 -28732.98,E2 -28732.98} C_VEL
LIN {X 0,Y 59.194,Z 523.872,A -85,B 0,C 180,E1 -28741.324,E2 -28741.324} C_VEL
LIN {X 0,Y 57.147,Z 525.625,A -85,B 0,C 180,E1 -28748.739,E2 -28748.739} C_VEL
LIN {X 0,Y 57.034,Z 526.684,A -85,B 0,C 180,E1 -28754.604,E2 -28754.604} C_VEL
LIN {X 0,Y 57.388,Z 526.96,A -85,B 0,C 180,E1 -28756.526,E2 -28756.526} C_VEL
LIN {X 0,Y 60.109,Z 527.957,A -85,B 0,C 180,E1 -28764.93,E2 -28764.93} C_VEL
LIN {X 0,Y 65.024,Z 528.325,A -85,B 0,C 180,E1 -28774.384,E2 -28774.384} C_VEL
LIN {X 0,Y 73.074,Z 527.453,A -85,B 0,C 180,E1 -28784.106,E2 -28784.106} C_VEL
LIN {X 0,Y 79.867,Z 525.869,A -85,B 0,C 180,E1 -28789.863,E2 -28789.863} C_VEL
LIN {X 0,Y 88.872,Z 522.917,A -85,B 0,C 180,E1 -28795.464,E2 -28795.464} C_VEL
LIN {X 0,Y 98.52,Z 518.705,A -85,B 0,C 180,E1 -28800,E2 -28800} C_VEL
LIN {X 0,Y 103.724,Z 515.984,A -85,B 0,C 180,E1 -28801.993,E2 -28801.993} C_VEL
LIN {X 0,Y 105.571,Z 514.899,A -85,B 0,C 180,E1 -28803.064,E2 -28803.064} C_VEL
LIN {X 0,Y 106.039,Z 514.569,A -85,B 0,C 180,E1 -28803.8,E2 -28803.8} C_VEL
LIN {X 0,Y 107.396,Z 513.451,A -85,B 0,C 180,E1 -28807.52,E2 -28807.52} C_VEL
LIN {X 0,Y 107.134,Z 513.551,A -85,B 0,C 180,E1 -28811.35,E2 -28811.35} C_VEL
LIN {X 0,Y 106.657,Z 514.085,A -85,B 0,C 180,E1 -28815.282,E2 -28815.282} C_VEL
LIN {X 0,Y 106.054,Z 515.049,A -85,B 0,C 180,E1 -28819.35,E2 -28819.35} C_VEL
LIN {X 0,Y 104.408,Z 517.291,A -85,B 0,C 180,E1 -28824.817,E2 -28824.817} C_VEL
LIN {X 0,Y 102.134,Z 518.918,A -85,B 0,C 180,E1 -28826.549,E2 -28826.549} C_VEL
LIN {X 0,Y 99.414,Z 520.585,A -85,B 0,C 180,E1 -28827.911,E2 -28827.911} C_VEL
LIN {X 0,Y 90.791,Z 524.996,A -85,B 0,C 180,E1 -28831.625,E2 -28831.625} C_VEL
LIN {X 0,Y 80.039,Z 529.389,A -85,B 0,C 180,E1 -28837.789,E2 -28837.789} C_VEL
LIN {X 0,Y 70.561,Z 532.271,A -85,B 0,C 180,E1 -28845.796,E2 -28845.796} C_VEL
LIN {X 0,Y 62.859,Z 533.641,A -85,B 0,C 180,E1 -28856.01,E2 -28856.01} C_VEL
LIN {X 0,Y 57.928,Z 533.621,A -85,B 0,C 180,E1 -28868.655,E2 -28868.655} C_VEL
LIN {X 0,Y 56.063,Z 532.144,A -85,B 0,C 180,E1 -28882.797,E2 -28882.797} C_VEL
LIN {X 0,Y 56.352,Z 530.811,A -85,B 0,C 180,E1 -28889.998,E2 -28889.998} C_VEL
LIN {X 0,Y 56.392,Z 527.819,A -85,B 0,C 180,E1 -28900.772,E2 -28900.772} C_VEL
LIN {X 0,Y 58.116,Z 523.737,A -85,B 0,C 180,E1 -28911.27,E2 -28911.27} C_VEL
LIN {X 0,Y 62.256,Z 517.463,A -85,B 0,C 180,E1 -28922.424,E2 -28922.424} C_VEL
LIN {X 0,Y 67.406,Z 510.614,A -85,B 0,C 180,E1 -28930.663,E2 -28930.663} C_VEL
LIN {X 0,Y 73.535,Z 502.269,A -85,B 0,C 180,E1 -28937.476,E2 -28937.476} C_VEL
LIN {X 0,Y 76.055,Z 496.448,A -85,B 0,C 180,E1 -28941.759,E2 -28941.759} C_VEL
LIN {X 0,Y 79.413,Z 486.73,A -85,B 0,C 180,E1 -28947.928,E2 -28947.928} C_VEL
LIN {X 0,Y 80.74,Z 482.129,A -85,B 0,C 180,E1 -28950.507,E2 -28950.507} C_VEL
LIN {X 0,Y 80.519,Z 477.416,A -85,B 0,C 180,E1 -28954.125,E2 -28954.125} C_VEL
LIN {X 0,Y 79.792,Z 471.071,A -85,B 0,C 180,E1 -28959.371,E2 -28959.371} C_VEL
LIN {X 0,Y 78.867,Z 465.441,A -85,B 0,C 180,E1 -28964.495,E2 -28964.495} C_VEL
LIN {X 0,Y 78.162,Z 461.714,A -85,B 0,C 180,E1 -28968.328,E2 -28968.328} C_VEL
LIN {X 0,Y 77.133,Z 458.995,A -85,B 0,C 180,E1 -28972.145,E2 -28972.145} C_VEL
LIN {X 0,Y 75.358,Z 454.78,A -85,B 0,C 180,E1 -28980.001,E2 -28980.001} C_VEL
LIN {X 0,Y 73.652,Z 452.097,A -85,B 0,C 180,E1 -28991.003,E2 -28991.003} C_VEL
LIN {X 0,Y 73.33,Z 451.884,A -85,B 0,C 180,E1 -28996.71,E2 -28996.71} C_VEL
LIN {X 0,Y 73.171,Z 452.803,A -85,B 0,C 180,E1 -29002.595,E2 -29002.595} C_VEL
LIN {X 0,Y 74.665,Z 455.363,A -85,B 0,C 180,E1 -29014.386,E2 -29014.386} C_VEL
LIN {X 0,Y 76.341,Z 459.384,A -85,B 0,C 180,E1 -29022.571,E2 -29022.571} C_VEL
LIN {X 0,Y 78.183,Z 464.176,A -85,B 0,C 180,E1 -29029.83,E2 -29029.83} C_VEL
LIN {X 0,Y 79.522,Z 468.313,A -85,B 0,C 180,E1 -29034.837,E2 -29034.837} C_VEL
LIN {X 0,Y 80.866,Z 473.482,A -85,B 0,C 180,E1 -29040.355,E2 -29040.355} C_VEL
LIN {X 0,Y 82.093,Z 479.377,A -85,B 0,C 180,E1 -29046.027,E2 -29046.027} C_VEL
LIN {X 0,Y 82.24,Z 482.55,A -85,B 0,C 180,E1 -29048.724,E2 -29048.724} C_VEL
LIN {X 0,Y 81.668,Z 484.383,A -85,B 0,C 180,E1 -29049.867,E2 -29049.867} C_VEL
LIN {X 0,Y 75.213,Z 494.185,A -85,B 0,C 180,E1 -29055.112,E2 -29055.112} C_VEL
LIN {X 0,Y 69.332,Z 502.262,A -85,B 0,C 180,E1 -29061.256,E2 -29061.256} C_VEL
LIN {X 0,Y 64.363,Z 508.902,A -85,B 0,C 180,E1 -29068.437,E2 -29068.437} C_VEL
LIN {X 0,Y 60.406,Z 514.37,A -85,B 0,C 180,E1 -29076.683,E2 -29076.683} C_VEL
LIN {X 0,Y 57.098,Z 519.654,A -85,B 0,C 180,E1 -29087.919,E2 -29087.919} C_VEL
LIN {X 0,Y 55.653,Z 523.649,A -85,B 0,C 180,E1 -29100.341,E2 -29100.341} C_VEL
LIN {X 0,Y 56.412,Z 526.161,A -85,B 0,C 180,E1 -29111.625,E2 -29111.625} C_VEL
LIN {X 0,Y 57.388,Z 526.96,A -85,B 0,C 180,E1 -29116.526,E2 -29116.526} C_VEL
LIN {X 0,Y 58.377,Z 527.757,A -85,B 0,C 180,E1 -29122.226,E2 -29122.226} C_VEL
LIN {X 0,Y 59.458,Z 528.497,A -85,B 0,C 180,E1 -29131.783,E2 -29131.783} C_VEL
LIN {X 0,Y 61.295,Z 528.717,A -85,B 0,C 180,E1 -29139.144,E2 -29139.144} C_VEL
LIN {X 0,Y 63.965,Z 528.582,A -85,B 0,C 180,E1 -29143.989,E2 -29143.989} C_VEL
LIN {X 0,Y 65.166,Z 528.468,A -85,B 0,C 180,E1 -29145.381,E2 -29145.381} C_VEL
LIN {X 0,Y 71.191,Z 527.547,A -85,B 0,C 180,E1 -29150.824,E2 -29150.824} C_VEL
LIN {X 0,Y 80.917,Z 525.166,A -85,B 0,C 180,E1 -29157.231,E2 -29157.231} C_VEL
LIN {X 0,Y 91.428,Z 521.443,A -85,B 0,C 180,E1 -29162.151,E2 -29162.151} C_VEL
LIN {X 0,Y 98.752,Z 518.115,A -85,B 0,C 180,E1 -29164.896,E2 -29164.896} C_VEL
LIN {X 0,Y 101.122,Z 516.834,A -85,B 0,C 180,E1 -29167.99,E2 -29167.99} C_VEL
LIN {X 0,Y 100.704,Z 517.1,A -85,B 0,C 180,E1 -29172.302,E2 -29172.302} C_VEL
LIN {X 0,Y 100.144,Z 517.737,A -85,B 0,C 180,E1 -29176.303,E2 -29176.303} C_VEL
LIN {X 0,Y 99.183,Z 518.931,A -85,B 0,C 180,E1 -29180.75,E2 -29180.75} C_VEL
LIN {X 0,Y 98.705,Z 519.452,A -85,B 0,C 180,E1 -29182.237,E2 -29182.237} C_VEL
LIN {X 0,Y 96.244,Z 520.965,A -85,B 0,C 180,E1 -29184.107,E2 -29184.107} C_VEL
LIN {X 0,Y 90.282,Z 523.901,A -85,B 0,C 180,E1 -29186.463,E2 -29186.463} C_VEL
LIN {X 0,Y 81.431,Z 527.479,A -85,B 0,C 180,E1 -29190.337,E2 -29190.337} C_VEL
LIN {X 0,Y 70.608,Z 530.89,A -85,B 0,C 180,E1 -29197.223,E2 -29197.223} C_VEL
LIN {X 0,Y 61.135,Z 532.81,A -85,B 0,C 180,E1 -29206.389,E2 -29206.389} C_VEL
LIN {X 0,Y 53.81,Z 533.329,A -85,B 0,C 180,E1 -29218.503,E2 -29218.503} C_VEL
LIN {X 0,Y 49.732,Z 532.411,A -85,B 0,C 180,E1 -29233.581,E2 -29233.581} C_VEL
LIN {X 0,Y 49.284,Z 529.99,A -85,B 0,C 180,E1 -29249.998,E2 -29249.998} C_VEL
LIN {X 0,Y 49.441,Z 526.844,A -85,B 0,C 180,E1 -29262.309,E2 -29262.309} C_VEL
LIN {X 0,Y 51.537,Z 522.596,A -85,B 0,C 180,E1 -29274.146,E2 -29274.146} C_VEL
LIN {X 0,Y 56.389,Z 516.141,A -85,B 0,C 180,E1 -29286.297,E2 -29286.297} C_VEL
LIN {X 0,Y 62.173,Z 509.02,A -85,B 0,C 180,E1 -29294.947,E2 -29294.947} C_VEL
LIN {X 0,Y 67.466,Z 502.344,A -85,B 0,C 180,E1 -29300.555,E2 -29300.555} C_VEL
LIN {X 0,Y 69.596,Z 498.158,A -85,B 0,C 180,E1 -29303.884,E2 -29303.884} C_VEL
LIN {X 0,Y 73.111,Z 489.651,A -85,B 0,C 180,E1 -29309.895,E2 -29309.895} C_VEL
LIN {X 0,Y 75.067,Z 483.792,A -85,B 0,C 180,E1 -29313.596,E2 -29313.596} C_VEL
LIN {X 0,Y 74.831,Z 476.797,A -85,B 0,C 180,E1 -29319.908,E2 -29319.908} C_VEL
LIN {X 0,Y 74.315,Z 470.291,A -85,B 0,C 180,E1 -29326.325,E2 -29326.325} C_VEL
LIN {X 0,Y 73.886,Z 466.717,A -85,B 0,C 180,E1 -29330.419,E2 -29330.419} C_VEL
LIN {X 0,Y 72.522,Z 462.768,A -85,B 0,C 180,E1 -29337.223,E2 -29337.223} C_VEL
LIN {X 0,Y 72.153,Z 461.381,A -85,B 0,C 180,E1 -29340.001,E2 -29340.001} C_VEL
LIN {X 0,Y 70.715,Z 458.553,A -85,B 0,C 180,E1 -29351.466,E2 -29351.466} C_VEL
LIN {X 0,Y 70.348,Z 458.542,A -85,B 0,C 180,E1 -29357.441,E2 -29357.441} C_VEL
LIN {X 0,Y 70.623,Z 460.792,A -85,B 0,C 180,E1 -29369.84,E2 -29369.84} C_VEL
LIN {X 0,Y 71.48,Z 462.751,A -85,B 0,C 180,E1 -29376.153,E2 -29376.153} C_VEL
LIN {X 0,Y 72.594,Z 465.791,A -85,B 0,C 180,E1 -29382.664,E2 -29382.664} C_VEL
LIN {X 0,Y 73.877,Z 470.099,A -85,B 0,C 180,E1 -29389.558,E2 -29389.558} C_VEL
LIN {X 0,Y 75.015,Z 474.975,A -85,B 0,C 180,E1 -29395.799,E2 -29395.799} C_VEL
LIN {X 0,Y 75.953,Z 480.933,A -85,B 0,C 180,E1 -29402.443,E2 -29402.443} C_VEL
LIN {X 0,Y 76.338,Z 483.854,A -85,B 0,C 180,E1 -29405.527,E2 -29405.527} C_VEL
LIN {X 0,Y 75.86,Z 485.552,A -85,B 0,C 180,E1 -29406.815,E2 -29406.815} C_VEL
LIN {X 0,Y 68.998,Z 495.254,A -85,B 0,C 180,E1 -29412.209,E2 -29412.209} C_VEL
LIN {X 0,Y 62.713,Z 503.239,A -85,B 0,C 180,E1 -29418.692,E2 -29418.692} C_VEL
LIN {X 0,Y 57.783,Z 509.334,A -85,B 0,C 180,E1 -29425.883,E2 -29425.883} C_VEL
LIN {X 0,Y 53.925,Z 514.161,A -85,B 0,C 180,E1 -29433.738,E2 -29433.738} C_VEL
LIN {X 0,Y 50.189,Z 519.609,A -85,B 0,C 180,E1 -29446.265,E2 -29446.265} C_VEL
LIN {X 0,Y 48.571,Z 523.593,A -85,B 0,C 180,E1 -29459.75,E2 -29459.75} C_VEL
LIN {X 0,Y 49.822,Z 526.659,A -85,B 0,C 180,E1 -29475.144,E2 -29475.144} C_VEL
LIN {X 0,Y 53.944,Z 528.337,A -85,B 0,C 180,E1 -29488.591,E2 -29488.591} C_VEL
LIN {X 0,Y 60.214,Z 528.791,A -85,B 0,C 180,E1 -29499.503,E2 -29499.503} C_VEL
LIN {X 0,Y 65.166,Z 528.468,A -85,B 0,C 180,E1 -29505.381,E2 -29505.381} C_VEL
LIN {X 0,Y 68.633,Z 528.127,A -85,B 0,C 180,E1 -29509.468,E2 -29509.468} C_VEL
LIN {X 0,Y 73.697,Z 527.089,A -85,B 0,C 180,E1 -29516.291,E2 -29516.291} C_VEL
LIN {X 0,Y 79.584,Z 525.394,A -85,B 0,C 180,E1 -29522.118,E2 -29522.118} C_VEL
LIN {X 0,Y 84.097,Z 523.976,A -85,B 0,C 180,E1 -29524.595,E2 -29524.595} C_VEL
LIN {X 0,Y 92.148,Z 520.957,A -85,B 0,C 180,E1 -29527.48,E2 -29527.48} C_VEL
LIN {X 0,Y 94.337,Z 520.055,A -85,B 0,C 180,E1 -29528.568,E2 -29528.568} C_VEL
LIN {X 0,Y 94.006,Z 520.379,A -85,B 0,C 180,E1 -29533.617,E2 -29533.617} C_VEL
LIN {X 0,Y 92.936,Z 521.475,A -85,B 0,C 180,E1 -29539.117,E2 -29539.117} C_VEL
LIN {X 0,Y 90.476,Z 522.781,A -85,B 0,C 180,E1 -29541.23,E2 -29541.23} C_VEL
LIN {X 0,Y 78.081,Z 527.559,A -85,B 0,C 180,E1 -29545.83,E2 -29545.83} C_VEL
LIN {X 0,Y 66.531,Z 530.735,A -85,B 0,C 180,E1 -29552.318,E2 -29552.318} C_VEL
LIN {X 0,Y 56.19,Z 532.49,A -85,B 0,C 180,E1 -29561.369,E2 -29561.369} C_VEL
LIN {X 0,Y 47.871,Z 532.814,A -85,B 0,C 180,E1 -29574.036,E2 -29574.036} C_VEL
LIN {X 0,Y 42.968,Z 531.71,A -85,B 0,C 180,E1 -29590.903,E2 -29590.903} C_VEL
LIN {X 0,Y 42.18,Z 529.384,A -85,B 0,C 180,E1 -29608.6,E2 -29608.6} C_VEL
LIN {X 0,Y 42.528,Z 525.849,A -85,B 0,C 180,E1 -29624.35,E2 -29624.35} C_VEL
LIN {X 0,Y 45.137,Z 521.442,A -85,B 0,C 180,E1 -29637.844,E2 -29637.844} C_VEL
LIN {X 0,Y 50.843,Z 514.733,A -85,B 0,C 180,E1 -29651.037,E2 -29651.037} C_VEL
LIN {X 0,Y 57.35,Z 507.407,A -85,B 0,C 180,E1 -29659.985,E2 -29659.985} C_VEL
LIN {X 0,Y 62.136,Z 501.684,A -85,B 0,C 180,E1 -29664.804,E2 -29664.804} C_VEL
LIN {X 0,Y 65.654,Z 494.897,A -85,B 0,C 180,E1 -29670.424,E2 -29670.424} C_VEL
LIN {X 0,Y 69.259,Z 486.772,A -85,B 0,C 180,E1 -29676.053,E2 -29676.053} C_VEL
LIN {X 0,Y 69.579,Z 480.456,A -85,B 0,C 180,E1 -29682.361,E2 -29682.361} C_VEL
LIN {X 0,Y 69.627,Z 474.985,A -85,B 0,C 180,E1 -29688.354,E2 -29688.354} C_VEL
LIN {X 0,Y 69.529,Z 472.58,A -85,B 0,C 180,E1 -29691.28,E2 -29691.28} C_VEL
LIN {X 0,Y 69.251,Z 470.713,A -85,B 0,C 180,E1 -29694.176,E2 -29694.176} C_VEL
LIN {X 0,Y 68.546,Z 467.816,A -85,B 0,C 180,E1 -29700.001,E2 -29700.001} C_VEL
LIN {X 0,Y 67.782,Z 466.086,A -85,B 0,C 180,E1 -29705.952,E2 -29705.952} C_VEL
LIN {X 0,Y 67.404,Z 464.874,A -85,B 0,C 180,E1 -29712.037,E2 -29712.037} C_VEL
LIN {X 0,Y 66.912,Z 465.139,A -85,B 0,C 180,E1 -29719.045,E2 -29719.045} C_VEL
LIN {X 0,Y 66.786,Z 466.065,A -85,B 0,C 180,E1 -29724.894,E2 -29724.894} C_VEL
LIN {X 0,Y 67.416,Z 468.115,A -85,B 0,C 180,E1 -29733.494,E2 -29733.494} C_VEL
